Fanuc TP program (LS listing): FM171157.ls

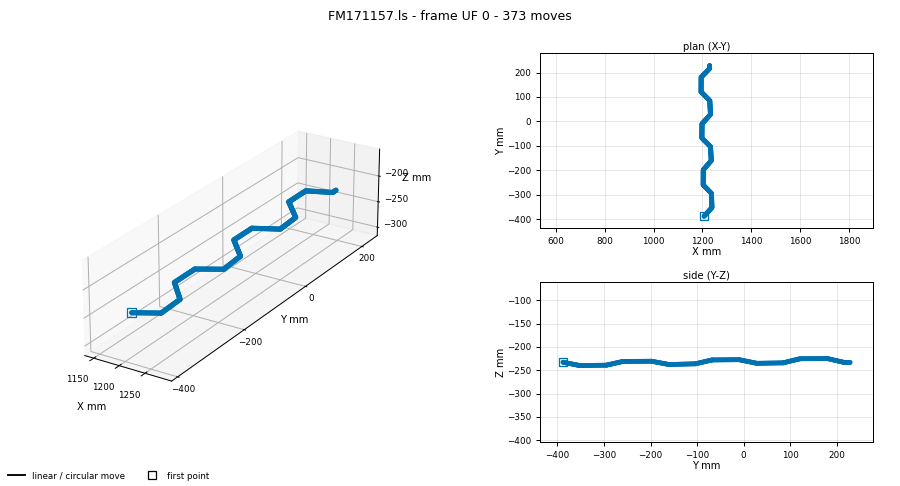
[picture p0: tool path of FM171157.ls in frame UF 0, 373 of 373 moves have a stored position in this frame; points joined in program order, loops and branches not executed]
/PROG  FM171157
/ATTR
OWNER		= MNEDITOR;
COMMENT		= "Auto FANUC move";
PROG_SIZE	= 0;
CREATE		= DATE 26-05-06  TIME 17:11:57;
MODIFIED	= DATE 26-05-06  TIME 17:11:57;
FILE_NAME	= ;
VERSION		= 0;
LINE_COUNT	= 378;
MEMORY_SIZE	= 0;
PROTECT		= READ_WRITE;
TCD:  STACK_SIZE	= 0,
      TASK_PRIORITY	= 50,
      TIME_SLICE	= 0,
      BUSY_LAMP_OFF	= 0,
      ABORT_REQUEST	= 0,
      PAUSE_REQUEST	= 0;
DEFAULT_GROUP	= 1,*,*,*,*;
CONTROL_CODE	= 00000000 00000000;
/MN
   1:  UFRAME_NUM=0 ;
   2:  UTOOL_NUM=1 ;
   3:  R[93]=10 ;
   4:  L P[1] 7mm/sec FINE ;
   5:  L P[2] 7mm/sec CNT50 ;
   6:  L P[3] 7mm/sec CNT50 ;
   7:  L P[4] 7mm/sec CNT50 ;
   8:  L P[5] 7mm/sec CNT50 ;
   9:  L P[6] 7mm/sec CNT50 ;
  10:  L P[7] 7mm/sec CNT50 ;
  11:  L P[8] 7mm/sec CNT50 ;
  12:  L P[9] 7mm/sec CNT50 ;
  13:  L P[10] 7mm/sec CNT50 ;
  14:  L P[11] 7mm/sec CNT50 ;
  15:  L P[12] 7mm/sec CNT50 ;
  16:  L P[13] 7mm/sec CNT50 ;
  17:  L P[14] 7mm/sec CNT50 ;
  18:  L P[15] 7mm/sec CNT50 ;
  19:  L P[16] 7mm/sec CNT50 ;
  20:  L P[17] 7mm/sec CNT50 ;
  21:  L P[18] 7mm/sec CNT50 ;
  22:  L P[19] 7mm/sec CNT50 ;
  23:  L P[20] 7mm/sec CNT50 ;
  24:  L P[21] 7mm/sec CNT50 ;
  25:  L P[22] 7mm/sec CNT50 ;
  26:  L P[23] 7mm/sec CNT50 ;
  27:  L P[24] 7mm/sec CNT50 ;
  28:  L P[25] 7mm/sec CNT50 ;
  29:  L P[26] 7mm/sec CNT50 ;
  30:  L P[27] 7mm/sec CNT50 ;
  31:  L P[28] 7mm/sec CNT50 ;
  32:  L P[29] 7mm/sec CNT50 ;
  33:  L P[30] 7mm/sec CNT50 ;
  34:  L P[31] 7mm/sec CNT50 ;
  35:  L P[32] 7mm/sec CNT50 ;
  36:  L P[33] 7mm/sec CNT50 ;
  37:  L P[34] 7mm/sec CNT50 ;
  38:  L P[35] 7mm/sec CNT50 ;
  39:  L P[36] 7mm/sec CNT50 ;
  40:  L P[37] 7mm/sec CNT50 ;
  41:  L P[38] 7mm/sec CNT50 ;
  42:  L P[39] 7mm/sec CNT50 ;
  43:  L P[40] 7mm/sec CNT50 ;
  44:  L P[41] 7mm/sec CNT50 ;
  45:  L P[42] 7mm/sec CNT50 ;
  46:  L P[43] 7mm/sec CNT50 ;
  47:  L P[44] 7mm/sec CNT50 ;
  48:  L P[45] 7mm/sec CNT50 ;
  49:  L P[46] 7mm/sec CNT50 ;
  50:  L P[47] 7mm/sec CNT50 ;
  51:  L P[48] 7mm/sec CNT50 ;
  52:  L P[49] 7mm/sec CNT50 ;
  53:  L P[50] 7mm/sec CNT50 ;
  54:  L P[51] 7mm/sec CNT50 ;
  55:  L P[52] 7mm/sec CNT50 ;
  56:  L P[53] 7mm/sec CNT50 ;
  57:  L P[54] 7mm/sec CNT50 ;
  58:  L P[55] 7mm/sec CNT50 ;
  59:  L P[56] 7mm/sec CNT50 ;
  60:  L P[57] 7mm/sec CNT50 ;
  61:  L P[58] 7mm/sec CNT50 ;
  62:  L P[59] 7mm/sec CNT50 ;
  63:  L P[60] 7mm/sec CNT50 ;
  64:  L P[61] 7mm/sec CNT50 ;
  65:  L P[62] 7mm/sec CNT50 ;
  66:  L P[63] 7mm/sec CNT50 ;
  67:  L P[64] 7mm/sec CNT50 ;
  68:  L P[65] 7mm/sec CNT50 ;
  69:  L P[66] 7mm/sec CNT50 ;
  70:  L P[67] 7mm/sec CNT50 ;
  71:  L P[68] 7mm/sec CNT50 ;
  72:  L P[69] 7mm/sec CNT50 ;
  73:  L P[70] 7mm/sec CNT50 ;
  74:  L P[71] 7mm/sec CNT50 ;
  75:  L P[72] 7mm/sec CNT50 ;
  76:  L P[73] 7mm/sec CNT50 ;
  77:  L P[74] 7mm/sec CNT50 ;
  78:  L P[75] 7mm/sec CNT50 ;
  79:  L P[76] 7mm/sec CNT50 ;
  80:  L P[77] 7mm/sec CNT50 ;
  81:  L P[78] 7mm/sec CNT50 ;
  82:  L P[79] 7mm/sec CNT50 ;
  83:  L P[80] 7mm/sec CNT50 ;
  84:  L P[81] 7mm/sec CNT50 ;
  85:  L P[82] 7mm/sec CNT50 ;
  86:  L P[83] 7mm/sec CNT50 ;
  87:  L P[84] 7mm/sec CNT50 ;
  88:  L P[85] 7mm/sec CNT50 ;
  89:  L P[86] 7mm/sec CNT50 ;
  90:  L P[87] 7mm/sec CNT50 ;
  91:  L P[88] 7mm/sec CNT50 ;
  92:  L P[89] 7mm/sec CNT50 ;
  93:  L P[90] 7mm/sec CNT50 ;
  94:  L P[91] 7mm/sec CNT50 ;
  95:  L P[92] 7mm/sec CNT50 ;
  96:  L P[93] 7mm/sec CNT50 ;
  97:  L P[94] 7mm/sec CNT50 ;
  98:  L P[95] 7mm/sec CNT50 ;
  99:  L P[96] 7mm/sec CNT50 ;
 100:  L P[97] 7mm/sec CNT50 ;
 101:  L P[98] 7mm/sec CNT50 ;
 102:  L P[99] 7mm/sec CNT50 ;
 103:  L P[100] 7mm/sec CNT50 ;
 104:  L P[101] 7mm/sec CNT50 ;
 105:  L P[102] 7mm/sec CNT50 ;
 106:  L P[103] 7mm/sec CNT50 ;
 107:  L P[104] 7mm/sec CNT50 ;
 108:  L P[105] 7mm/sec CNT50 ;
 109:  L P[106] 7mm/sec CNT50 ;
 110:  L P[107] 7mm/sec CNT50 ;
 111:  L P[108] 7mm/sec CNT50 ;
 112:  L P[109] 7mm/sec CNT50 ;
 113:  L P[110] 7mm/sec CNT50 ;
 114:  L P[111] 7mm/sec CNT50 ;
 115:  L P[112] 7mm/sec CNT50 ;
 116:  L P[113] 7mm/sec CNT50 ;
 117:  L P[114] 7mm/sec CNT50 ;
 118:  L P[115] 7mm/sec CNT50 ;
 119:  L P[116] 7mm/sec CNT50 ;
 120:  L P[117] 7mm/sec CNT50 ;
 121:  L P[118] 7mm/sec CNT50 ;
 122:  L P[119] 7mm/sec CNT50 ;
 123:  L P[120] 7mm/sec CNT50 ;
 124:  L P[121] 7mm/sec CNT50 ;
 125:  L P[122] 7mm/sec CNT50 ;
 126:  L P[123] 7mm/sec CNT50 ;
 127:  L P[124] 7mm/sec CNT50 ;
 128:  L P[125] 7mm/sec CNT50 ;
 129:  L P[126] 7mm/sec CNT50 ;
 130:  L P[127] 7mm/sec CNT50 ;
 131:  L P[128] 7mm/sec CNT50 ;
 132:  L P[129] 7mm/sec CNT50 ;
 133:  L P[130] 7mm/sec CNT50 ;
 134:  L P[131] 7mm/sec CNT50 ;
 135:  L P[132] 7mm/sec CNT50 ;
 136:  L P[133] 7mm/sec CNT50 ;
 137:  L P[134] 7mm/sec CNT50 ;
 138:  L P[135] 7mm/sec CNT50 ;
 139:  L P[136] 7mm/sec CNT50 ;
 140:  L P[137] 7mm/sec CNT50 ;
 141:  L P[138] 7mm/sec CNT50 ;
 142:  L P[139] 7mm/sec CNT50 ;
 143:  L P[140] 7mm/sec CNT50 ;
 144:  L P[141] 7mm/sec CNT50 ;
 145:  L P[142] 7mm/sec CNT50 ;
 146:  L P[143] 7mm/sec CNT50 ;
 147:  L P[144] 7mm/sec CNT50 ;
 148:  L P[145] 7mm/sec CNT50 ;
 149:  L P[146] 7mm/sec CNT50 ;
 150:  L P[147] 7mm/sec CNT50 ;
 151:  L P[148] 7mm/sec CNT50 ;
 152:  L P[149] 7mm/sec CNT50 ;
 153:  L P[150] 7mm/sec CNT50 ;
 154:  L P[151] 7mm/sec CNT50 ;
 155:  L P[152] 7mm/sec CNT50 ;
 156:  L P[153] 7mm/sec CNT50 ;
 157:  L P[154] 7mm/sec CNT50 ;
 158:  L P[155] 7mm/sec CNT50 ;
 159:  L P[156] 7mm/sec CNT50 ;
 160:  L P[157] 7mm/sec CNT50 ;
 161:  L P[158] 7mm/sec CNT50 ;
 162:  L P[159] 7mm/sec CNT50 ;
 163:  L P[160] 7mm/sec CNT50 ;
 164:  L P[161] 7mm/sec CNT50 ;
 165:  L P[162] 7mm/sec CNT50 ;
 166:  L P[163] 7mm/sec CNT50 ;
 167:  L P[164] 7mm/sec CNT50 ;
 168:  L P[165] 7mm/sec CNT50 ;
 169:  L P[166] 7mm/sec CNT50 ;
 170:  L P[167] 7mm/sec CNT50 ;
 171:  L P[168] 7mm/sec CNT50 ;
 172:  L P[169] 7mm/sec CNT50 ;
 173:  L P[170] 7mm/sec CNT50 ;
 174:  L P[171] 7mm/sec CNT50 ;
 175:  L P[172] 7mm/sec CNT50 ;
 176:  L P[173] 7mm/sec CNT50 ;
 177:  L P[174] 7mm/sec CNT50 ;
 178:  L P[175] 7mm/sec CNT50 ;
 179:  L P[176] 7mm/sec CNT50 ;
 180:  L P[177] 7mm/sec CNT50 ;
 181:  L P[178] 7mm/sec CNT50 ;
 182:  L P[179] 7mm/sec CNT50 ;
 183:  L P[180] 7mm/sec CNT50 ;
 184:  L P[181] 7mm/sec CNT50 ;
 185:  L P[182] 7mm/sec CNT50 ;
 186:  L P[183] 7mm/sec CNT50 ;
 187:  L P[184] 7mm/sec CNT50 ;
 188:  L P[185] 7mm/sec CNT50 ;
 189:  L P[186] 7mm/sec CNT50 ;
 190:  L P[187] 7mm/sec CNT50 ;
 191:  L P[188] 7mm/sec CNT50 ;
 192:  L P[189] 7mm/sec CNT50 ;
 193:  L P[190] 7mm/sec CNT50 ;
 194:  L P[191] 7mm/sec CNT50 ;
 195:  L P[192] 7mm/sec CNT50 ;
 196:  L P[193] 7mm/sec CNT50 ;
 197:  L P[194] 7mm/sec CNT50 ;
 198:  L P[195] 7mm/sec CNT50 ;
 199:  L P[196] 7mm/sec CNT50 ;
 200:  L P[197] 7mm/sec CNT50 ;
 201:  L P[198] 7mm/sec CNT50 ;
 202:  L P[199] 7mm/sec CNT50 ;
 203:  L P[200] 7mm/sec CNT50 ;
 204:  L P[201] 7mm/sec CNT50 ;
 205:  L P[202] 7mm/sec CNT50 ;
 206:  L P[203] 7mm/sec CNT50 ;
 207:  L P[204] 7mm/sec CNT50 ;
 208:  L P[205] 7mm/sec CNT50 ;
 209:  L P[206] 7mm/sec CNT50 ;
 210:  L P[207] 7mm/sec CNT50 ;
 211:  L P[208] 7mm/sec CNT50 ;
 212:  L P[209] 7mm/sec CNT50 ;
 213:  L P[210] 7mm/sec CNT50 ;
 214:  L P[211] 7mm/sec CNT50 ;
 215:  L P[212] 7mm/sec CNT50 ;
 216:  L P[213] 7mm/sec CNT50 ;
 217:  L P[214] 7mm/sec CNT50 ;
 218:  L P[215] 7mm/sec CNT50 ;
 219:  L P[216] 7mm/sec CNT50 ;
 220:  L P[217] 7mm/sec CNT50 ;
 221:  L P[218] 7mm/sec CNT50 ;
 222:  L P[219] 7mm/sec CNT50 ;
 223:  L P[220] 7mm/sec CNT50 ;
 224:  L P[221] 7mm/sec CNT50 ;
 225:  L P[222] 7mm/sec CNT50 ;
 226:  L P[223] 7mm/sec CNT50 ;
 227:  L P[224] 7mm/sec CNT50 ;
 228:  L P[225] 7mm/sec CNT50 ;
 229:  L P[226] 7mm/sec CNT50 ;
 230:  L P[227] 7mm/sec CNT50 ;
 231:  L P[228] 7mm/sec CNT50 ;
 232:  L P[229] 7mm/sec CNT50 ;
 233:  L P[230] 7mm/sec CNT50 ;
 234:  L P[231] 7mm/sec CNT50 ;
 235:  L P[232] 7mm/sec CNT50 ;
 236:  L P[233] 7mm/sec CNT50 ;
 237:  L P[234] 7mm/sec CNT50 ;
 238:  L P[235] 7mm/sec CNT50 ;
 239:  L P[236] 7mm/sec CNT50 ;
 240:  L P[237] 7mm/sec CNT50 ;
 241:  L P[238] 7mm/sec CNT50 ;
 242:  L P[239] 7mm/sec CNT50 ;
 243:  L P[240] 7mm/sec CNT50 ;
 244:  L P[241] 7mm/sec CNT50 ;
 245:  L P[242] 7mm/sec CNT50 ;
 246:  L P[243] 7mm/sec CNT50 ;
 247:  L P[244] 7mm/sec CNT50 ;
 248:  L P[245] 7mm/sec CNT50 ;
 249:  L P[246] 7mm/sec CNT50 ;
 250:  L P[247] 7mm/sec CNT50 ;
 251:  L P[248] 7mm/sec CNT50 ;
 252:  L P[249] 7mm/sec CNT50 ;
 253:  L P[250] 7mm/sec CNT50 ;
 254:  L P[251] 7mm/sec CNT50 ;
 255:  L P[252] 7mm/sec CNT50 ;
 256:  L P[253] 7mm/sec CNT50 ;
 257:  L P[254] 7mm/sec CNT50 ;
 258:  L P[255] 7mm/sec CNT50 ;
 259:  L P[256] 7mm/sec CNT50 ;
 260:  L P[257] 7mm/sec CNT50 ;
 261:  L P[258] 7mm/sec CNT50 ;
 262:  L P[259] 7mm/sec CNT50 ;
 263:  L P[260] 7mm/sec CNT50 ;
 264:  L P[261] 7mm/sec CNT50 ;
 265:  L P[262] 7mm/sec CNT50 ;
 266:  L P[263] 7mm/sec CNT50 ;
 267:  L P[264] 7mm/sec CNT50 ;
 268:  L P[265] 7mm/sec CNT50 ;
 269:  L P[266] 7mm/sec CNT50 ;
 270:  L P[267] 7mm/sec CNT50 ;
 271:  L P[268] 7mm/sec CNT50 ;
 272:  L P[269] 7mm/sec CNT50 ;
 273:  L P[270] 7mm/sec CNT50 ;
 274:  L P[271] 7mm/sec CNT50 ;
 275:  L P[272] 7mm/sec CNT50 ;
 276:  L P[273] 7mm/sec CNT50 ;
 277:  L P[274] 7mm/sec CNT50 ;
 278:  L P[275] 7mm/sec CNT50 ;
 279:  L P[276] 7mm/sec CNT50 ;
 280:  L P[277] 7mm/sec CNT50 ;
 281:  L P[278] 7mm/sec CNT50 ;
 282:  L P[279] 7mm/sec CNT50 ;
 283:  L P[280] 7mm/sec CNT50 ;
 284:  L P[281] 7mm/sec CNT50 ;
 285:  L P[282] 7mm/sec CNT50 ;
 286:  L P[283] 7mm/sec CNT50 ;
 287:  L P[284] 7mm/sec CNT50 ;
 288:  L P[285] 7mm/sec CNT50 ;
 289:  L P[286] 7mm/sec CNT50 ;
 290:  L P[287] 7mm/sec CNT50 ;
 291:  L P[288] 7mm/sec CNT50 ;
 292:  L P[289] 7mm/sec CNT50 ;
 293:  L P[290] 7mm/sec CNT50 ;
 294:  L P[291] 7mm/sec CNT50 ;
 295:  L P[292] 7mm/sec CNT50 ;
 296:  L P[293] 7mm/sec CNT50 ;
 297:  L P[294] 7mm/sec CNT50 ;
 298:  L P[295] 7mm/sec CNT50 ;
 299:  L P[296] 7mm/sec CNT50 ;
 300:  L P[297] 7mm/sec CNT50 ;
 301:  L P[298] 7mm/sec CNT50 ;
 302:  L P[299] 7mm/sec CNT50 ;
 303:  L P[300] 7mm/sec CNT50 ;
 304:  L P[301] 7mm/sec CNT50 ;
 305:  L P[302] 7mm/sec CNT50 ;
 306:  L P[303] 7mm/sec CNT50 ;
 307:  L P[304] 7mm/sec CNT50 ;
 308:  L P[305] 7mm/sec CNT50 ;
 309:  L P[306] 7mm/sec CNT50 ;
 310:  L P[307] 7mm/sec CNT50 ;
 311:  L P[308] 7mm/sec CNT50 ;
 312:  L P[309] 7mm/sec CNT50 ;
 313:  L P[310] 7mm/sec CNT50 ;
 314:  L P[311] 7mm/sec CNT50 ;
 315:  L P[312] 7mm/sec CNT50 ;
 316:  L P[313] 7mm/sec CNT50 ;
 317:  L P[314] 7mm/sec CNT50 ;
 318:  L P[315] 7mm/sec CNT50 ;
 319:  L P[316] 7mm/sec CNT50 ;
 320:  L P[317] 7mm/sec CNT50 ;
 321:  L P[318] 7mm/sec CNT50 ;
 322:  L P[319] 7mm/sec CNT50 ;
 323:  L P[320] 7mm/sec CNT50 ;
 324:  L P[321] 7mm/sec CNT50 ;
 325:  L P[322] 7mm/sec CNT50 ;
 326:  L P[323] 7mm/sec CNT50 ;
 327:  L P[324] 7mm/sec CNT50 ;
 328:  L P[325] 7mm/sec CNT50 ;
 329:  L P[326] 7mm/sec CNT50 ;
 330:  L P[327] 7mm/sec CNT50 ;
 331:  L P[328] 7mm/sec CNT50 ;
 332:  L P[329] 7mm/sec CNT50 ;
 333:  L P[330] 7mm/sec CNT50 ;
 334:  L P[331] 7mm/sec CNT50 ;
 335:  L P[332] 7mm/sec CNT50 ;
 336:  L P[333] 7mm/sec CNT50 ;
 337:  L P[334] 7mm/sec CNT50 ;
 338:  L P[335] 7mm/sec CNT50 ;
 339:  L P[336] 7mm/sec CNT50 ;
 340:  L P[337] 7mm/sec CNT50 ;
 341:  L P[338] 7mm/sec CNT50 ;
 342:  L P[339] 7mm/sec CNT50 ;
 343:  L P[340] 7mm/sec CNT50 ;
 344:  L P[341] 7mm/sec CNT50 ;
 345:  L P[342] 7mm/sec CNT50 ;
 346:  L P[343] 7mm/sec CNT50 ;
 347:  L P[344] 7mm/sec CNT50 ;
 348:  L P[345] 7mm/sec CNT50 ;
 349:  L P[346] 7mm/sec CNT50 ;
 350:  L P[347] 7mm/sec CNT50 ;
 351:  L P[348] 7mm/sec CNT50 ;
 352:  L P[349] 7mm/sec CNT50 ;
 353:  L P[350] 7mm/sec CNT50 ;
 354:  L P[351] 7mm/sec CNT50 ;
 355:  L P[352] 7mm/sec CNT50 ;
 356:  L P[353] 7mm/sec CNT50 ;
 357:  L P[354] 7mm/sec CNT50 ;
 358:  L P[355] 7mm/sec CNT50 ;
 359:  L P[356] 7mm/sec CNT50 ;
 360:  L P[357] 7mm/sec CNT50 ;
 361:  L P[358] 7mm/sec CNT50 ;
 362:  L P[359] 7mm/sec CNT50 ;
 363:  L P[360] 7mm/sec CNT50 ;
 364:  L P[361] 7mm/sec CNT50 ;
 365:  L P[362] 7mm/sec CNT50 ;
 366:  L P[363] 7mm/sec CNT50 ;
 367:  L P[364] 7mm/sec CNT50 ;
 368:  L P[365] 7mm/sec CNT50 ;
 369:  L P[366] 7mm/sec CNT50 ;
 370:  L P[367] 7mm/sec CNT50 ;
 371:  L P[368] 7mm/sec CNT50 ;
 372:  L P[369] 7mm/sec CNT50 ;
 373:  L P[370] 7mm/sec CNT50 ;
 374:  L P[371] 7mm/sec CNT50 ;
 375:  L P[372] 7mm/sec CNT50 ;
 376:  L P[373] 7mm/sec FINE ;
 377:  R[93]=1 ;
 378:  END ;
/POS
P[1]{
   GP1:
	UF : 0, UT : 1,		CONFIG : 'N U T, 0, 0, 0',
	X = 1206.347  mm,	Y = -388.199  mm,	Z = -232.788  mm,
	W = 0.000 deg,	P = 30.000 deg,	R = 160.000 deg
};
P[2]{
   GP1:
	UF : 0, UT : 1,		CONFIG : 'N U T, 0, 0, 0',
	X = 1207.673  mm,	Y = -386.730  mm,	Z = -233.078  mm,
	W = 0.000 deg,	P = 30.000 deg,	R = 160.000 deg
};
P[3]{
   GP1:
	UF : 0, UT : 1,		CONFIG : 'N U T, 0, 0, 0',
	X = 1208.999  mm,	Y = -385.261  mm,	Z = -233.367  mm,
	W = 0.000 deg,	P = 30.000 deg,	R = 160.000 deg
};
P[4]{
   GP1:
	UF : 0, UT : 1,		CONFIG : 'N U T, 0, 0, 0',
	X = 1210.325  mm,	Y = -383.791  mm,	Z = -233.656  mm,
	W = 0.000 deg,	P = 30.000 deg,	R = 160.000 deg
};
P[5]{
   GP1:
	UF : 0, UT : 1,		CONFIG : 'N U T, 0, 0, 0',
	X = 1211.651  mm,	Y = -382.322  mm,	Z = -233.946  mm,
	W = 0.000 deg,	P = 30.000 deg,	R = 160.000 deg
};
P[6]{
   GP1:
	UF : 0, UT : 1,		CONFIG : 'N U T, 0, 0, 0',
	X = 1212.977  mm,	Y = -380.853  mm,	Z = -234.235  mm,
	W = 0.000 deg,	P = 30.000 deg,	R = 160.000 deg
};
P[7]{
   GP1:
	UF : 0, UT : 1,		CONFIG : 'N U T, 0, 0, 0',
	X = 1214.303  mm,	Y = -379.384  mm,	Z = -234.524  mm,
	W = 0.000 deg,	P = 30.000 deg,	R = 160.000 deg
};
P[8]{
   GP1:
	UF : 0, UT : 1,		CONFIG : 'N U T, 0, 0, 0',
	X = 1215.629  mm,	Y = -377.915  mm,	Z = -234.814  mm,
	W = 0.000 deg,	P = 30.000 deg,	R = 160.000 deg
};
P[9]{
   GP1:
	UF : 0, UT : 1,		CONFIG : 'N U T, 0, 0, 0',
	X = 1216.955  mm,	Y = -376.446  mm,	Z = -235.103  mm,
	W = 0.000 deg,	P = 30.000 deg,	R = 160.000 deg
};
P[10]{
   GP1:
	UF : 0, UT : 1,		CONFIG : 'N U T, 0, 0, 0',
	X = 1218.281  mm,	Y = -374.977  mm,	Z = -235.392  mm,
	W = 0.000 deg,	P = 30.000 deg,	R = 160.000 deg
};
P[11]{
   GP1:
	UF : 0, UT : 1,		CONFIG : 'N U T, 0, 0, 0',
	X = 1219.607  mm,	Y = -373.508  mm,	Z = -235.682  mm,
	W = 0.000 deg,	P = 30.000 deg,	R = 160.000 deg
};
P[12]{
   GP1:
	UF : 0, UT : 1,		CONFIG : 'N U T, 0, 0, 0',
	X = 1220.933  mm,	Y = -372.039  mm,	Z = -235.971  mm,
	W = 0.000 deg,	P = 30.000 deg,	R = 160.000 deg
};
P[13]{
   GP1:
	UF : 0, UT : 1,		CONFIG : 'N U T, 0, 0, 0',
	X = 1222.258  mm,	Y = -370.570  mm,	Z = -236.260  mm,
	W = 0.000 deg,	P = 30.000 deg,	R = 160.000 deg
};
P[14]{
   GP1:
	UF : 0, UT : 1,		CONFIG : 'N U T, 0, 0, 0',
	X = 1223.584  mm,	Y = -369.101  mm,	Z = -236.549  mm,
	W = 0.000 deg,	P = 30.000 deg,	R = 160.000 deg
};
P[15]{
   GP1:
	UF : 0, UT : 1,		CONFIG : 'N U T, 0, 0, 0',
	X = 1224.910  mm,	Y = -367.632  mm,	Z = -236.839  mm,
	W = 0.000 deg,	P = 30.000 deg,	R = 160.000 deg
};
P[16]{
   GP1:
	UF : 0, UT : 1,		CONFIG : 'N U T, 0, 0, 0',
	X = 1226.236  mm,	Y = -366.163  mm,	Z = -237.128  mm,
	W = 0.000 deg,	P = 30.000 deg,	R = 160.000 deg
};
P[17]{
   GP1:
	UF : 0, UT : 1,		CONFIG : 'N U T, 0, 0, 0',
	X = 1227.562  mm,	Y = -364.694  mm,	Z = -237.417  mm,
	W = 0.000 deg,	P = 30.000 deg,	R = 160.000 deg
};
P[18]{
   GP1:
	UF : 0, UT : 1,		CONFIG : 'N U T, 0, 0, 0',
	X = 1228.888  mm,	Y = -363.225  mm,	Z = -237.707  mm,
	W = 0.000 deg,	P = 30.000 deg,	R = 160.000 deg
};
P[19]{
   GP1:
	UF : 0, UT : 1,		CONFIG : 'N U T, 0, 0, 0',
	X = 1230.214  mm,	Y = -361.756  mm,	Z = -237.996  mm,
	W = 0.000 deg,	P = 30.000 deg,	R = 160.000 deg
};
P[20]{
   GP1:
	UF : 0, UT : 1,		CONFIG : 'N U T, 0, 0, 0',
	X = 1231.540  mm,	Y = -360.287  mm,	Z = -238.285  mm,
	W = 0.000 deg,	P = 30.000 deg,	R = 160.000 deg
};
P[21]{
   GP1:
	UF : 0, UT : 1,		CONFIG : 'N U T, 0, 0, 0',
	X = 1232.866  mm,	Y = -358.818  mm,	Z = -238.575  mm,
	W = 0.000 deg,	P = 30.000 deg,	R = 164.342 deg
};
P[22]{
   GP1:
	UF : 0, UT : 1,		CONFIG : 'N U T, 0, 0, 0',
	X = 1234.192  mm,	Y = -357.349  mm,	Z = -238.864  mm,
	W = 0.000 deg,	P = 30.000 deg,	R = 168.685 deg
};
P[23]{
   GP1:
	UF : 0, UT : 1,		CONFIG : 'N U T, 0, 0, 0',
	X = 1235.518  mm,	Y = -355.880  mm,	Z = -239.153  mm,
	W = 0.000 deg,	P = 30.000 deg,	R = 173.027 deg
};
P[24]{
   GP1:
	UF : 0, UT : 1,		CONFIG : 'N U T, 0, 0, 0',
	X = 1236.844  mm,	Y = -354.410  mm,	Z = -239.443  mm,
	W = 0.000 deg,	P = 30.000 deg,	R = 177.369 deg
};
P[25]{
   GP1:
	UF : 0, UT : 1,		CONFIG : 'N U T, 0, 0, 0',
	X = 1238.170  mm,	Y = -352.941  mm,	Z = -239.732  mm,
	W = 0.000 deg,	P = 30.000 deg,	R = -178.289 deg
};
P[26]{
   GP1:
	UF : 0, UT : 1,		CONFIG : 'N U T, 0, 0, 0',
	X = 1238.798  mm,	Y = -352.246  mm,	Z = -239.869  mm,
	W = 0.000 deg,	P = 30.000 deg,	R = -178.289 deg
};
P[27]{
   GP1:
	UF : 0, UT : 1,		CONFIG : 'N U T, 0, 0, 0',
	X = 1238.766  mm,	Y = -351.193  mm,	Z = -239.854  mm,
	W = 0.000 deg,	P = 30.000 deg,	R = -178.289 deg
};
P[28]{
   GP1:
	UF : 0, UT : 1,		CONFIG : 'N U T, 0, 0, 0',
	X = 1238.706  mm,	Y = -349.194  mm,	Z = -239.826  mm,
	W = 0.000 deg,	P = 30.000 deg,	R = -178.289 deg
};
P[29]{
   GP1:
	UF : 0, UT : 1,		CONFIG : 'N U T, 0, 0, 0',
	X = 1238.647  mm,	Y = -347.195  mm,	Z = -239.798  mm,
	W = 0.000 deg,	P = 30.000 deg,	R = -178.289 deg
};
P[30]{
   GP1:
	UF : 0, UT : 1,		CONFIG : 'N U T, 0, 0, 0',
	X = 1238.587  mm,	Y = -345.197  mm,	Z = -239.769  mm,
	W = 0.000 deg,	P = 30.000 deg,	R = -178.289 deg
};
P[31]{
   GP1:
	UF : 0, UT : 1,		CONFIG : 'N U T, 0, 0, 0',
	X = 1238.527  mm,	Y = -343.198  mm,	Z = -239.741  mm,
	W = 0.000 deg,	P = 30.000 deg,	R = -178.289 deg
};
P[32]{
   GP1:
	UF : 0, UT : 1,		CONFIG : 'N U T, 0, 0, 0',
	X = 1238.468  mm,	Y = -341.199  mm,	Z = -239.713  mm,
	W = 0.000 deg,	P = 30.000 deg,	R = -178.289 deg
};
P[33]{
   GP1:
	UF : 0, UT : 1,		CONFIG : 'N U T, 0, 0, 0',
	X = 1238.408  mm,	Y = -339.200  mm,	Z = -239.685  mm,
	W = 0.000 deg,	P = 30.000 deg,	R = -178.289 deg
};
P[34]{
   GP1:
	UF : 0, UT : 1,		CONFIG : 'N U T, 0, 0, 0',
	X = 1238.348  mm,	Y = -337.201  mm,	Z = -239.656  mm,
	W = 0.000 deg,	P = 30.000 deg,	R = -178.289 deg
};
P[35]{
   GP1:
	UF : 0, UT : 1,		CONFIG : 'N U T, 0, 0, 0',
	X = 1238.288  mm,	Y = -335.202  mm,	Z = -239.628  mm,
	W = 0.000 deg,	P = 30.000 deg,	R = -178.289 deg
};
P[36]{
   GP1:
	UF : 0, UT : 1,		CONFIG : 'N U T, 0, 0, 0',
	X = 1238.229  mm,	Y = -333.203  mm,	Z = -239.600  mm,
	W = 0.000 deg,	P = 30.000 deg,	R = -178.289 deg
};
P[37]{
   GP1:
	UF : 0, UT : 1,		CONFIG : 'N U T, 0, 0, 0',
	X = 1238.169  mm,	Y = -331.204  mm,	Z = -239.572  mm,
	W = 0.000 deg,	P = 30.000 deg,	R = -178.289 deg
};
P[38]{
   GP1:
	UF : 0, UT : 1,		CONFIG : 'N U T, 0, 0, 0',
	X = 1238.109  mm,	Y = -329.205  mm,	Z = -239.543  mm,
	W = 0.000 deg,	P = 30.000 deg,	R = -178.289 deg
};
P[39]{
   GP1:
	UF : 0, UT : 1,		CONFIG : 'N U T, 0, 0, 0',
	X = 1238.049  mm,	Y = -327.206  mm,	Z = -239.515  mm,
	W = 0.000 deg,	P = 30.000 deg,	R = -178.289 deg
};
P[40]{
   GP1:
	UF : 0, UT : 1,		CONFIG : 'N U T, 0, 0, 0',
	X = 1237.990  mm,	Y = -325.207  mm,	Z = -239.487  mm,
	W = 0.000 deg,	P = 30.000 deg,	R = -178.289 deg
};
P[41]{
   GP1:
	UF : 0, UT : 1,		CONFIG : 'N U T, 0, 0, 0',
	X = 1237.930  mm,	Y = -323.209  mm,	Z = -239.459  mm,
	W = 0.000 deg,	P = 30.000 deg,	R = -178.289 deg
};
P[42]{
   GP1:
	UF : 0, UT : 1,		CONFIG : 'N U T, 0, 0, 0',
	X = 1237.870  mm,	Y = -321.210  mm,	Z = -239.431  mm,
	W = 0.000 deg,	P = 30.000 deg,	R = -178.289 deg
};
P[43]{
   GP1:
	UF : 0, UT : 1,		CONFIG : 'N U T, 0, 0, 0',
	X = 1237.811  mm,	Y = -319.211  mm,	Z = -239.402  mm,
	W = 0.000 deg,	P = 30.000 deg,	R = -178.289 deg
};
P[44]{
   GP1:
	UF : 0, UT : 1,		CONFIG : 'N U T, 0, 0, 0',
	X = 1237.751  mm,	Y = -317.212  mm,	Z = -239.374  mm,
	W = 0.000 deg,	P = 30.000 deg,	R = -178.289 deg
};
P[45]{
   GP1:
	UF : 0, UT : 1,		CONFIG : 'N U T, 0, 0, 0',
	X = 1237.691  mm,	Y = -315.213  mm,	Z = -239.346  mm,
	W = 0.000 deg,	P = 30.000 deg,	R = -178.289 deg
};
P[46]{
   GP1:
	UF : 0, UT : 1,		CONFIG : 'N U T, 0, 0, 0',
	X = 1237.631  mm,	Y = -313.214  mm,	Z = -239.318  mm,
	W = 0.000 deg,	P = 30.000 deg,	R = -178.289 deg
};
P[47]{
   GP1:
	UF : 0, UT : 1,		CONFIG : 'N U T, 0, 0, 0',
	X = 1237.572  mm,	Y = -311.215  mm,	Z = -239.289  mm,
	W = 0.000 deg,	P = 30.000 deg,	R = -178.289 deg
};
P[48]{
   GP1:
	UF : 0, UT : 1,		CONFIG : 'N U T, 0, 0, 0',
	X = 1237.512  mm,	Y = -309.216  mm,	Z = -239.261  mm,
	W = 0.000 deg,	P = 30.000 deg,	R = -178.289 deg
};
P[49]{
   GP1:
	UF : 0, UT : 1,		CONFIG : 'N U T, 0, 0, 0',
	X = 1237.452  mm,	Y = -307.217  mm,	Z = -239.233  mm,
	W = 0.000 deg,	P = 30.000 deg,	R = -178.289 deg
};
P[50]{
   GP1:
	UF : 0, UT : 1,		CONFIG : 'N U T, 0, 0, 0',
	X = 1237.393  mm,	Y = -305.218  mm,	Z = -239.205  mm,
	W = 0.000 deg,	P = 30.000 deg,	R = -178.289 deg
};
P[51]{
   GP1:
	UF : 0, UT : 1,		CONFIG : 'N U T, 0, 0, 0',
	X = 1237.333  mm,	Y = -303.219  mm,	Z = -239.177  mm,
	W = 0.000 deg,	P = 30.000 deg,	R = -172.704 deg
};
P[52]{
   GP1:
	UF : 0, UT : 1,		CONFIG : 'N U T, 0, 0, 0',
	X = 1237.273  mm,	Y = -301.221  mm,	Z = -239.148  mm,
	W = 0.000 deg,	P = 30.000 deg,	R = -169.047 deg
};
P[53]{
   GP1:
	UF : 0, UT : 1,		CONFIG : 'N U T, 0, 0, 0',
	X = 1237.213  mm,	Y = -299.222  mm,	Z = -239.120  mm,
	W = 0.000 deg,	P = 30.000 deg,	R = -165.389 deg
};
P[54]{
   GP1:
	UF : 0, UT : 1,		CONFIG : 'N U T, 0, 0, 0',
	X = 1237.154  mm,	Y = -297.223  mm,	Z = -239.092  mm,
	W = 0.000 deg,	P = 30.000 deg,	R = -161.731 deg
};
P[55]{
   GP1:
	UF : 0, UT : 1,		CONFIG : 'N U T, 0, 0, 0',
	X = 1237.094  mm,	Y = -295.224  mm,	Z = -239.064  mm,
	W = 0.000 deg,	P = 30.000 deg,	R = -160.000 deg
};
P[56]{
   GP1:
	UF : 0, UT : 1,		CONFIG : 'N U T, 0, 0, 0',
	X = 1237.079  mm,	Y = -294.716  mm,	Z = -239.056  mm,
	W = 0.000 deg,	P = 30.000 deg,	R = -160.000 deg
};
P[57]{
   GP1:
	UF : 0, UT : 1,		CONFIG : 'N U T, 0, 0, 0',
	X = 1236.053  mm,	Y = -293.659  mm,	Z = -238.818  mm,
	W = 0.000 deg,	P = 30.000 deg,	R = -160.000 deg
};
P[58]{
   GP1:
	UF : 0, UT : 1,		CONFIG : 'N U T, 0, 0, 0',
	X = 1234.678  mm,	Y = -292.243  mm,	Z = -238.498  mm,
	W = 0.000 deg,	P = 30.000 deg,	R = -160.000 deg
};
P[59]{
   GP1:
	UF : 0, UT : 1,		CONFIG : 'N U T, 0, 0, 0',
	X = 1233.303  mm,	Y = -290.826  mm,	Z = -238.177  mm,
	W = 0.000 deg,	P = 30.000 deg,	R = -160.000 deg
};
P[60]{
   GP1:
	UF : 0, UT : 1,		CONFIG : 'N U T, 0, 0, 0',
	X = 1231.928  mm,	Y = -289.409  mm,	Z = -237.857  mm,
	W = 0.000 deg,	P = 30.000 deg,	R = -160.000 deg
};
P[61]{
   GP1:
	UF : 0, UT : 1,		CONFIG : 'N U T, 0, 0, 0',
	X = 1230.553  mm,	Y = -287.992  mm,	Z = -237.537  mm,
	W = 0.000 deg,	P = 30.000 deg,	R = -160.000 deg
};
P[62]{
   GP1:
	UF : 0, UT : 1,		CONFIG : 'N U T, 0, 0, 0',
	X = 1229.179  mm,	Y = -286.575  mm,	Z = -237.217  mm,
	W = 0.000 deg,	P = 30.000 deg,	R = -160.000 deg
};
P[63]{
   GP1:
	UF : 0, UT : 1,		CONFIG : 'N U T, 0, 0, 0',
	X = 1227.804  mm,	Y = -285.159  mm,	Z = -236.897  mm,
	W = 0.000 deg,	P = 30.000 deg,	R = -160.000 deg
};
P[64]{
   GP1:
	UF : 0, UT : 1,		CONFIG : 'N U T, 0, 0, 0',
	X = 1226.429  mm,	Y = -283.742  mm,	Z = -236.577  mm,
	W = 0.000 deg,	P = 30.000 deg,	R = -160.000 deg
};
P[65]{
   GP1:
	UF : 0, UT : 1,		CONFIG : 'N U T, 0, 0, 0',
	X = 1225.054  mm,	Y = -282.325  mm,	Z = -236.257  mm,
	W = 0.000 deg,	P = 30.000 deg,	R = -160.000 deg
};
P[66]{
   GP1:
	UF : 0, UT : 1,		CONFIG : 'N U T, 0, 0, 0',
	X = 1223.679  mm,	Y = -280.908  mm,	Z = -235.937  mm,
	W = 0.000 deg,	P = 30.000 deg,	R = -160.000 deg
};
P[67]{
   GP1:
	UF : 0, UT : 1,		CONFIG : 'N U T, 0, 0, 0',
	X = 1222.304  mm,	Y = -279.491  mm,	Z = -235.617  mm,
	W = 0.000 deg,	P = 30.000 deg,	R = -160.000 deg
};
P[68]{
   GP1:
	UF : 0, UT : 1,		CONFIG : 'N U T, 0, 0, 0',
	X = 1220.929  mm,	Y = -278.075  mm,	Z = -235.297  mm,
	W = 0.000 deg,	P = 30.000 deg,	R = -160.000 deg
};
P[69]{
   GP1:
	UF : 0, UT : 1,		CONFIG : 'N U T, 0, 0, 0',
	X = 1219.554  mm,	Y = -276.658  mm,	Z = -234.977  mm,
	W = 0.000 deg,	P = 30.000 deg,	R = -160.000 deg
};
P[70]{
   GP1:
	UF : 0, UT : 1,		CONFIG : 'N U T, 0, 0, 0',
	X = 1218.180  mm,	Y = -275.241  mm,	Z = -234.656  mm,
	W = 0.000 deg,	P = 30.000 deg,	R = -160.000 deg
};
P[71]{
   GP1:
	UF : 0, UT : 1,		CONFIG : 'N U T, 0, 0, 0',
	X = 1216.805  mm,	Y = -273.824  mm,	Z = -234.336  mm,
	W = 0.000 deg,	P = 30.000 deg,	R = -160.000 deg
};
P[72]{
   GP1:
	UF : 0, UT : 1,		CONFIG : 'N U T, 0, 0, 0',
	X = 1215.430  mm,	Y = -272.408  mm,	Z = -234.016  mm,
	W = 0.000 deg,	P = 30.000 deg,	R = -160.000 deg
};
P[73]{
   GP1:
	UF : 0, UT : 1,		CONFIG : 'N U T, 0, 0, 0',
	X = 1214.055  mm,	Y = -270.991  mm,	Z = -233.696  mm,
	W = 0.000 deg,	P = 30.000 deg,	R = -160.000 deg
};
P[74]{
   GP1:
	UF : 0, UT : 1,		CONFIG : 'N U T, 0, 0, 0',
	X = 1212.680  mm,	Y = -269.574  mm,	Z = -233.376  mm,
	W = 0.000 deg,	P = 30.000 deg,	R = -160.000 deg
};
P[75]{
   GP1:
	UF : 0, UT : 1,		CONFIG : 'N U T, 0, 0, 0',
	X = 1211.305  mm,	Y = -268.157  mm,	Z = -233.056  mm,
	W = 0.000 deg,	P = 30.000 deg,	R = -160.000 deg
};
P[76]{
   GP1:
	UF : 0, UT : 1,		CONFIG : 'N U T, 0, 0, 0',
	X = 1209.930  mm,	Y = -266.740  mm,	Z = -232.736  mm,
	W = 0.000 deg,	P = 30.000 deg,	R = -160.000 deg
};
P[77]{
   GP1:
	UF : 0, UT : 1,		CONFIG : 'N U T, 0, 0, 0',
	X = 1208.555  mm,	Y = -265.324  mm,	Z = -232.416  mm,
	W = 0.000 deg,	P = 30.000 deg,	R = -167.071 deg
};
P[78]{
   GP1:
	UF : 0, UT : 1,		CONFIG : 'N U T, 0, 0, 0',
	X = 1207.181  mm,	Y = -263.907  mm,	Z = -232.096  mm,
	W = 0.000 deg,	P = 30.000 deg,	R = -171.121 deg
};
P[79]{
   GP1:
	UF : 0, UT : 1,		CONFIG : 'N U T, 0, 0, 0',
	X = 1205.806  mm,	Y = -262.490  mm,	Z = -231.776  mm,
	W = 0.000 deg,	P = 30.000 deg,	R = -175.171 deg
};
P[80]{
   GP1:
	UF : 0, UT : 1,		CONFIG : 'N U T, 0, 0, 0',
	X = 1204.431  mm,	Y = -261.073  mm,	Z = -231.455  mm,
	W = 0.000 deg,	P = 30.000 deg,	R = -179.220 deg
};
P[81]{
   GP1:
	UF : 0, UT : 1,		CONFIG : 'N U T, 0, 0, 0',
	X = 1203.056  mm,	Y = -259.657  mm,	Z = -231.135  mm,
	W = 0.000 deg,	P = 30.000 deg,	R = 179.752 deg
};
P[82]{
   GP1:
	UF : 0, UT : 1,		CONFIG : 'N U T, 0, 0, 0',
	X = 1202.896  mm,	Y = -259.492  mm,	Z = -231.098  mm,
	W = 0.000 deg,	P = 30.000 deg,	R = 179.752 deg
};
P[83]{
   GP1:
	UF : 0, UT : 1,		CONFIG : 'N U T, 0, 0, 0',
	X = 1202.904  mm,	Y = -257.724  mm,	Z = -231.083  mm,
	W = 0.000 deg,	P = 30.000 deg,	R = 179.752 deg
};
P[84]{
   GP1:
	UF : 0, UT : 1,		CONFIG : 'N U T, 0, 0, 0',
	X = 1202.912  mm,	Y = -255.725  mm,	Z = -231.067  mm,
	W = 0.000 deg,	P = 30.000 deg,	R = 179.752 deg
};
P[85]{
   GP1:
	UF : 0, UT : 1,		CONFIG : 'N U T, 0, 0, 0',
	X = 1202.921  mm,	Y = -253.725  mm,	Z = -231.050  mm,
	W = 0.000 deg,	P = 30.000 deg,	R = 179.752 deg
};
P[86]{
   GP1:
	UF : 0, UT : 1,		CONFIG : 'N U T, 0, 0, 0',
	X = 1202.930  mm,	Y = -251.725  mm,	Z = -231.033  mm,
	W = 0.000 deg,	P = 30.000 deg,	R = 179.752 deg
};
P[87]{
   GP1:
	UF : 0, UT : 1,		CONFIG : 'N U T, 0, 0, 0',
	X = 1202.938  mm,	Y = -249.725  mm,	Z = -231.016  mm,
	W = 0.000 deg,	P = 30.000 deg,	R = 179.752 deg
};
P[88]{
   GP1:
	UF : 0, UT : 1,		CONFIG : 'N U T, 0, 0, 0',
	X = 1202.947  mm,	Y = -247.725  mm,	Z = -230.999  mm,
	W = 0.000 deg,	P = 30.000 deg,	R = 179.752 deg
};
P[89]{
   GP1:
	UF : 0, UT : 1,		CONFIG : 'N U T, 0, 0, 0',
	X = 1202.956  mm,	Y = -245.725  mm,	Z = -230.983  mm,
	W = 0.000 deg,	P = 30.000 deg,	R = 179.752 deg
};
P[90]{
   GP1:
	UF : 0, UT : 1,		CONFIG : 'N U T, 0, 0, 0',
	X = 1202.965  mm,	Y = -243.725  mm,	Z = -230.966  mm,
	W = 0.000 deg,	P = 30.000 deg,	R = 179.752 deg
};
P[91]{
   GP1:
	UF : 0, UT : 1,		CONFIG : 'N U T, 0, 0, 0',
	X = 1202.973  mm,	Y = -241.725  mm,	Z = -230.949  mm,
	W = 0.000 deg,	P = 30.000 deg,	R = 179.752 deg
};
P[92]{
   GP1:
	UF : 0, UT : 1,		CONFIG : 'N U T, 0, 0, 0',
	X = 1202.982  mm,	Y = -239.725  mm,	Z = -230.932  mm,
	W = 0.000 deg,	P = 30.000 deg,	R = 179.752 deg
};
P[93]{
   GP1:
	UF : 0, UT : 1,		CONFIG : 'N U T, 0, 0, 0',
	X = 1202.991  mm,	Y = -237.725  mm,	Z = -230.916  mm,
	W = 0.000 deg,	P = 30.000 deg,	R = 179.752 deg
};
P[94]{
   GP1:
	UF : 0, UT : 1,		CONFIG : 'N U T, 0, 0, 0',
	X = 1202.999  mm,	Y = -235.725  mm,	Z = -230.899  mm,
	W = 0.000 deg,	P = 30.000 deg,	R = 179.752 deg
};
P[95]{
   GP1:
	UF : 0, UT : 1,		CONFIG : 'N U T, 0, 0, 0',
	X = 1203.008  mm,	Y = -233.726  mm,	Z = -230.882  mm,
	W = 0.000 deg,	P = 30.000 deg,	R = 179.752 deg
};
P[96]{
   GP1:
	UF : 0, UT : 1,		CONFIG : 'N U T, 0, 0, 0',
	X = 1203.017  mm,	Y = -231.726  mm,	Z = -230.865  mm,
	W = 0.000 deg,	P = 30.000 deg,	R = 179.752 deg
};
P[97]{
   GP1:
	UF : 0, UT : 1,		CONFIG : 'N U T, 0, 0, 0',
	X = 1203.025  mm,	Y = -229.726  mm,	Z = -230.848  mm,
	W = 0.000 deg,	P = 30.000 deg,	R = 179.752 deg
};
P[98]{
   GP1:
	UF : 0, UT : 1,		CONFIG : 'N U T, 0, 0, 0',
	X = 1203.034  mm,	Y = -227.726  mm,	Z = -230.832  mm,
	W = 0.000 deg,	P = 30.000 deg,	R = 179.752 deg
};
P[99]{
   GP1:
	UF : 0, UT : 1,		CONFIG : 'N U T, 0, 0, 0',
	X = 1203.043  mm,	Y = -225.726  mm,	Z = -230.815  mm,
	W = 0.000 deg,	P = 30.000 deg,	R = 179.752 deg
};
P[100]{
   GP1:
	UF : 0, UT : 1,		CONFIG : 'N U T, 0, 0, 0',
	X = 1203.051  mm,	Y = -223.726  mm,	Z = -230.798  mm,
	W = 0.000 deg,	P = 30.000 deg,	R = 179.752 deg
};
P[101]{
   GP1:
	UF : 0, UT : 1,		CONFIG : 'N U T, 0, 0, 0',
	X = 1203.060  mm,	Y = -221.726  mm,	Z = -230.781  mm,
	W = 0.000 deg,	P = 30.000 deg,	R = 179.752 deg
};
P[102]{
   GP1:
	UF : 0, UT : 1,		CONFIG : 'N U T, 0, 0, 0',
	X = 1203.069  mm,	Y = -219.726  mm,	Z = -230.765  mm,
	W = 0.000 deg,	P = 30.000 deg,	R = 179.752 deg
};
P[103]{
   GP1:
	UF : 0, UT : 1,		CONFIG : 'N U T, 0, 0, 0',
	X = 1203.077  mm,	Y = -217.726  mm,	Z = -230.748  mm,
	W = 0.000 deg,	P = 30.000 deg,	R = 179.752 deg
};
P[104]{
   GP1:
	UF : 0, UT : 1,		CONFIG : 'N U T, 0, 0, 0',
	X = 1203.086  mm,	Y = -215.726  mm,	Z = -230.731  mm,
	W = 0.000 deg,	P = 30.000 deg,	R = 179.752 deg
};
P[105]{
   GP1:
	UF : 0, UT : 1,		CONFIG : 'N U T, 0, 0, 0',
	X = 1203.095  mm,	Y = -213.726  mm,	Z = -230.714  mm,
	W = 0.000 deg,	P = 30.000 deg,	R = 179.752 deg
};
P[106]{
   GP1:
	UF : 0, UT : 1,		CONFIG : 'N U T, 0, 0, 0',
	X = 1203.103  mm,	Y = -211.726  mm,	Z = -230.698  mm,
	W = 0.000 deg,	P = 30.000 deg,	R = 179.752 deg
};
P[107]{
   GP1:
	UF : 0, UT : 1,		CONFIG : 'N U T, 0, 0, 0',
	X = 1203.112  mm,	Y = -209.727  mm,	Z = -230.681  mm,
	W = 0.000 deg,	P = 30.000 deg,	R = 179.752 deg
};
P[108]{
   GP1:
	UF : 0, UT : 1,		CONFIG : 'N U T, 0, 0, 0',
	X = 1203.121  mm,	Y = -207.727  mm,	Z = -230.664  mm,
	W = 0.000 deg,	P = 30.000 deg,	R = 179.752 deg
};
P[109]{
   GP1:
	UF : 0, UT : 1,		CONFIG : 'N U T, 0, 0, 0',
	X = 1203.129  mm,	Y = -205.727  mm,	Z = -230.647  mm,
	W = 0.000 deg,	P = 30.000 deg,	R = 172.310 deg
};
P[110]{
   GP1:
	UF : 0, UT : 1,		CONFIG : 'N U T, 0, 0, 0',
	X = 1203.138  mm,	Y = -203.727  mm,	Z = -230.630  mm,
	W = 0.000 deg,	P = 30.000 deg,	R = 168.360 deg
};
P[111]{
   GP1:
	UF : 0, UT : 1,		CONFIG : 'N U T, 0, 0, 0',
	X = 1203.147  mm,	Y = -201.727  mm,	Z = -230.614  mm,
	W = 0.000 deg,	P = 30.000 deg,	R = 164.410 deg
};
P[112]{
   GP1:
	UF : 0, UT : 1,		CONFIG : 'N U T, 0, 0, 0',
	X = 1203.155  mm,	Y = -199.727  mm,	Z = -230.597  mm,
	W = 0.000 deg,	P = 30.000 deg,	R = 160.459 deg
};
P[113]{
   GP1:
	UF : 0, UT : 1,		CONFIG : 'N U T, 0, 0, 0',
	X = 1203.162  mm,	Y = -198.274  mm,	Z = -230.585  mm,
	W = 0.000 deg,	P = 30.000 deg,	R = 160.000 deg
};
P[114]{
   GP1:
	UF : 0, UT : 1,		CONFIG : 'N U T, 0, 0, 0',
	X = 1203.516  mm,	Y = -197.865  mm,	Z = -230.661  mm,
	W = 0.000 deg,	P = 30.000 deg,	R = 160.000 deg
};
P[115]{
   GP1:
	UF : 0, UT : 1,		CONFIG : 'N U T, 0, 0, 0',
	X = 1204.813  mm,	Y = -196.368  mm,	Z = -230.942  mm,
	W = 0.000 deg,	P = 30.000 deg,	R = 160.000 deg
};
P[116]{
   GP1:
	UF : 0, UT : 1,		CONFIG : 'N U T, 0, 0, 0',
	X = 1206.109  mm,	Y = -194.871  mm,	Z = -231.223  mm,
	W = 0.000 deg,	P = 30.000 deg,	R = 160.000 deg
};
P[117]{
   GP1:
	UF : 0, UT : 1,		CONFIG : 'N U T, 0, 0, 0',
	X = 1207.406  mm,	Y = -193.374  mm,	Z = -231.503  mm,
	W = 0.000 deg,	P = 30.000 deg,	R = 160.000 deg
};
P[118]{
   GP1:
	UF : 0, UT : 1,		CONFIG : 'N U T, 0, 0, 0',
	X = 1208.702  mm,	Y = -191.878  mm,	Z = -231.784  mm,
	W = 0.000 deg,	P = 30.000 deg,	R = 160.000 deg
};
P[119]{
   GP1:
	UF : 0, UT : 1,		CONFIG : 'N U T, 0, 0, 0',
	X = 1209.999  mm,	Y = -190.381  mm,	Z = -232.065  mm,
	W = 0.000 deg,	P = 30.000 deg,	R = 160.000 deg
};
P[120]{
   GP1:
	UF : 0, UT : 1,		CONFIG : 'N U T, 0, 0, 0',
	X = 1211.295  mm,	Y = -188.884  mm,	Z = -232.345  mm,
	W = 0.000 deg,	P = 30.000 deg,	R = 160.000 deg
};
P[121]{
   GP1:
	UF : 0, UT : 1,		CONFIG : 'N U T, 0, 0, 0',
	X = 1212.592  mm,	Y = -187.387  mm,	Z = -232.626  mm,
	W = 0.000 deg,	P = 30.000 deg,	R = 160.000 deg
};
P[122]{
   GP1:
	UF : 0, UT : 1,		CONFIG : 'N U T, 0, 0, 0',
	X = 1213.888  mm,	Y = -185.891  mm,	Z = -232.907  mm,
	W = 0.000 deg,	P = 30.000 deg,	R = 160.000 deg
};
P[123]{
   GP1:
	UF : 0, UT : 1,		CONFIG : 'N U T, 0, 0, 0',
	X = 1215.185  mm,	Y = -184.394  mm,	Z = -233.187  mm,
	W = 0.000 deg,	P = 30.000 deg,	R = 160.000 deg
};
P[124]{
   GP1:
	UF : 0, UT : 1,		CONFIG : 'N U T, 0, 0, 0',
	X = 1216.481  mm,	Y = -182.897  mm,	Z = -233.468  mm,
	W = 0.000 deg,	P = 30.000 deg,	R = 160.000 deg
};
P[125]{
   GP1:
	UF : 0, UT : 1,		CONFIG : 'N U T, 0, 0, 0',
	X = 1217.778  mm,	Y = -181.400  mm,	Z = -233.749  mm,
	W = 0.000 deg,	P = 30.000 deg,	R = 160.000 deg
};
P[126]{
   GP1:
	UF : 0, UT : 1,		CONFIG : 'N U T, 0, 0, 0',
	X = 1219.074  mm,	Y = -179.903  mm,	Z = -234.029  mm,
	W = 0.000 deg,	P = 30.000 deg,	R = 160.000 deg
};
P[127]{
   GP1:
	UF : 0, UT : 1,		CONFIG : 'N U T, 0, 0, 0',
	X = 1220.371  mm,	Y = -178.407  mm,	Z = -234.310  mm,
	W = 0.000 deg,	P = 30.000 deg,	R = 160.000 deg
};
P[128]{
   GP1:
	UF : 0, UT : 1,		CONFIG : 'N U T, 0, 0, 0',
	X = 1221.667  mm,	Y = -176.910  mm,	Z = -234.591  mm,
	W = 0.000 deg,	P = 30.000 deg,	R = 160.000 deg
};
P[129]{
   GP1:
	UF : 0, UT : 1,		CONFIG : 'N U T, 0, 0, 0',
	X = 1222.964  mm,	Y = -175.413  mm,	Z = -234.871  mm,
	W = 0.000 deg,	P = 30.000 deg,	R = 160.000 deg
};
P[130]{
   GP1:
	UF : 0, UT : 1,		CONFIG : 'N U T, 0, 0, 0',
	X = 1224.260  mm,	Y = -173.916  mm,	Z = -235.152  mm,
	W = 0.000 deg,	P = 30.000 deg,	R = 160.000 deg
};
P[131]{
   GP1:
	UF : 0, UT : 1,		CONFIG : 'N U T, 0, 0, 0',
	X = 1225.557  mm,	Y = -172.420  mm,	Z = -235.433  mm,
	W = 0.000 deg,	P = 30.000 deg,	R = 160.000 deg
};
P[132]{
   GP1:
	UF : 0, UT : 1,		CONFIG : 'N U T, 0, 0, 0',
	X = 1226.853  mm,	Y = -170.923  mm,	Z = -235.713  mm,
	W = 0.000 deg,	P = 30.000 deg,	R = 160.000 deg
};
P[133]{
   GP1:
	UF : 0, UT : 1,		CONFIG : 'N U T, 0, 0, 0',
	X = 1228.150  mm,	Y = -169.426  mm,	Z = -235.994  mm,
	W = 0.000 deg,	P = 30.000 deg,	R = 160.000 deg
};
P[134]{
   GP1:
	UF : 0, UT : 1,		CONFIG : 'N U T, 0, 0, 0',
	X = 1229.446  mm,	Y = -167.929  mm,	Z = -236.275  mm,
	W = 0.000 deg,	P = 30.000 deg,	R = 161.238 deg
};
P[135]{
   GP1:
	UF : 0, UT : 1,		CONFIG : 'N U T, 0, 0, 0',
	X = 1230.743  mm,	Y = -166.432  mm,	Z = -236.555  mm,
	W = 0.000 deg,	P = 30.000 deg,	R = 165.761 deg
};
P[136]{
   GP1:
	UF : 0, UT : 1,		CONFIG : 'N U T, 0, 0, 0',
	X = 1232.039  mm,	Y = -164.936  mm,	Z = -236.836  mm,
	W = 0.000 deg,	P = 30.000 deg,	R = 170.284 deg
};
P[137]{
   GP1:
	UF : 0, UT : 1,		CONFIG : 'N U T, 0, 0, 0',
	X = 1233.336  mm,	Y = -163.439  mm,	Z = -237.117  mm,
	W = 0.000 deg,	P = 30.000 deg,	R = 174.808 deg
};
P[138]{
   GP1:
	UF : 0, UT : 1,		CONFIG : 'N U T, 0, 0, 0',
	X = 1234.632  mm,	Y = -161.942  mm,	Z = -237.397  mm,
	W = 0.000 deg,	P = 30.000 deg,	R = 179.331 deg
};
P[139]{
   GP1:
	UF : 0, UT : 1,		CONFIG : 'N U T, 0, 0, 0',
	X = 1235.891  mm,	Y = -160.489  mm,	Z = -237.670  mm,
	W = 0.000 deg,	P = 30.000 deg,	R = -177.384 deg
};
P[140]{
   GP1:
	UF : 0, UT : 1,		CONFIG : 'N U T, 0, 0, 0',
	X = 1235.889  mm,	Y = -160.431  mm,	Z = -237.669  mm,
	W = 0.000 deg,	P = 30.000 deg,	R = -177.384 deg
};
P[141]{
   GP1:
	UF : 0, UT : 1,		CONFIG : 'N U T, 0, 0, 0',
	X = 1235.797  mm,	Y = -158.434  mm,	Z = -237.616  mm,
	W = 0.000 deg,	P = 30.000 deg,	R = -177.384 deg
};
P[142]{
   GP1:
	UF : 0, UT : 1,		CONFIG : 'N U T, 0, 0, 0',
	X = 1235.706  mm,	Y = -156.436  mm,	Z = -237.563  mm,
	W = 0.000 deg,	P = 30.000 deg,	R = -177.384 deg
};
P[143]{
   GP1:
	UF : 0, UT : 1,		CONFIG : 'N U T, 0, 0, 0',
	X = 1235.615  mm,	Y = -154.439  mm,	Z = -237.510  mm,
	W = 0.000 deg,	P = 30.000 deg,	R = -177.384 deg
};
P[144]{
   GP1:
	UF : 0, UT : 1,		CONFIG : 'N U T, 0, 0, 0',
	X = 1235.524  mm,	Y = -152.442  mm,	Z = -237.457  mm,
	W = 0.000 deg,	P = 30.000 deg,	R = -177.384 deg
};
P[145]{
   GP1:
	UF : 0, UT : 1,		CONFIG : 'N U T, 0, 0, 0',
	X = 1235.432  mm,	Y = -150.445  mm,	Z = -237.404  mm,
	W = 0.000 deg,	P = 30.000 deg,	R = -177.384 deg
};
P[146]{
   GP1:
	UF : 0, UT : 1,		CONFIG : 'N U T, 0, 0, 0',
	X = 1235.341  mm,	Y = -148.448  mm,	Z = -237.351  mm,
	W = 0.000 deg,	P = 30.000 deg,	R = -177.384 deg
};
P[147]{
   GP1:
	UF : 0, UT : 1,		CONFIG : 'N U T, 0, 0, 0',
	X = 1235.250  mm,	Y = -146.450  mm,	Z = -237.299  mm,
	W = 0.000 deg,	P = 30.000 deg,	R = -177.384 deg
};
P[148]{
   GP1:
	UF : 0, UT : 1,		CONFIG : 'N U T, 0, 0, 0',
	X = 1235.158  mm,	Y = -144.453  mm,	Z = -237.246  mm,
	W = 0.000 deg,	P = 30.000 deg,	R = -177.384 deg
};
P[149]{
   GP1:
	UF : 0, UT : 1,		CONFIG : 'N U T, 0, 0, 0',
	X = 1235.067  mm,	Y = -142.456  mm,	Z = -237.193  mm,
	W = 0.000 deg,	P = 30.000 deg,	R = -177.384 deg
};
P[150]{
   GP1:
	UF : 0, UT : 1,		CONFIG : 'N U T, 0, 0, 0',
	X = 1234.976  mm,	Y = -140.459  mm,	Z = -237.140  mm,
	W = 0.000 deg,	P = 30.000 deg,	R = -177.384 deg
};
P[151]{
   GP1:
	UF : 0, UT : 1,		CONFIG : 'N U T, 0, 0, 0',
	X = 1234.885  mm,	Y = -138.461  mm,	Z = -237.087  mm,
	W = 0.000 deg,	P = 30.000 deg,	R = -177.384 deg
};
P[152]{
   GP1:
	UF : 0, UT : 1,		CONFIG : 'N U T, 0, 0, 0',
	X = 1234.793  mm,	Y = -136.464  mm,	Z = -237.034  mm,
	W = 0.000 deg,	P = 30.000 deg,	R = -177.384 deg
};
P[153]{
   GP1:
	UF : 0, UT : 1,		CONFIG : 'N U T, 0, 0, 0',
	X = 1234.702  mm,	Y = -134.467  mm,	Z = -236.981  mm,
	W = 0.000 deg,	P = 30.000 deg,	R = -177.384 deg
};
P[154]{
   GP1:
	UF : 0, UT : 1,		CONFIG : 'N U T, 0, 0, 0',
	X = 1234.611  mm,	Y = -132.470  mm,	Z = -236.929  mm,
	W = 0.000 deg,	P = 30.000 deg,	R = -177.384 deg
};
P[155]{
   GP1:
	UF : 0, UT : 1,		CONFIG : 'N U T, 0, 0, 0',
	X = 1234.520  mm,	Y = -130.473  mm,	Z = -236.876  mm,
	W = 0.000 deg,	P = 30.000 deg,	R = -177.384 deg
};
P[156]{
   GP1:
	UF : 0, UT : 1,		CONFIG : 'N U T, 0, 0, 0',
	X = 1234.428  mm,	Y = -128.475  mm,	Z = -236.823  mm,
	W = 0.000 deg,	P = 30.000 deg,	R = -177.384 deg
};
P[157]{
   GP1:
	UF : 0, UT : 1,		CONFIG : 'N U T, 0, 0, 0',
	X = 1234.337  mm,	Y = -126.478  mm,	Z = -236.770  mm,
	W = 0.000 deg,	P = 30.000 deg,	R = -177.384 deg
};
P[158]{
   GP1:
	UF : 0, UT : 1,		CONFIG : 'N U T, 0, 0, 0',
	X = 1234.246  mm,	Y = -124.481  mm,	Z = -236.717  mm,
	W = 0.000 deg,	P = 30.000 deg,	R = -177.384 deg
};
P[159]{
   GP1:
	UF : 0, UT : 1,		CONFIG : 'N U T, 0, 0, 0',
	X = 1234.155  mm,	Y = -122.484  mm,	Z = -236.664  mm,
	W = 0.000 deg,	P = 30.000 deg,	R = -177.384 deg
};
P[160]{
   GP1:
	UF : 0, UT : 1,		CONFIG : 'N U T, 0, 0, 0',
	X = 1234.063  mm,	Y = -120.487  mm,	Z = -236.611  mm,
	W = 0.000 deg,	P = 30.000 deg,	R = -177.384 deg
};
P[161]{
   GP1:
	UF : 0, UT : 1,		CONFIG : 'N U T, 0, 0, 0',
	X = 1233.972  mm,	Y = -118.489  mm,	Z = -236.559  mm,
	W = 0.000 deg,	P = 30.000 deg,	R = -177.384 deg
};
P[162]{
   GP1:
	UF : 0, UT : 1,		CONFIG : 'N U T, 0, 0, 0',
	X = 1233.881  mm,	Y = -116.492  mm,	Z = -236.506  mm,
	W = 0.000 deg,	P = 30.000 deg,	R = -177.384 deg
};
P[163]{
   GP1:
	UF : 0, UT : 1,		CONFIG : 'N U T, 0, 0, 0',
	X = 1233.790  mm,	Y = -114.495  mm,	Z = -236.453  mm,
	W = 0.000 deg,	P = 30.000 deg,	R = -177.384 deg
};
P[164]{
   GP1:
	UF : 0, UT : 1,		CONFIG : 'N U T, 0, 0, 0',
	X = 1233.698  mm,	Y = -112.498  mm,	Z = -236.400  mm,
	W = 0.000 deg,	P = 30.000 deg,	R = -173.807 deg
};
P[165]{
   GP1:
	UF : 0, UT : 1,		CONFIG : 'N U T, 0, 0, 0',
	X = 1233.607  mm,	Y = -110.500  mm,	Z = -236.347  mm,
	W = 0.000 deg,	P = 30.000 deg,	R = -170.330 deg
};
P[166]{
   GP1:
	UF : 0, UT : 1,		CONFIG : 'N U T, 0, 0, 0',
	X = 1233.516  mm,	Y = -108.503  mm,	Z = -236.294  mm,
	W = 0.000 deg,	P = 30.000 deg,	R = -166.853 deg
};
P[167]{
   GP1:
	UF : 0, UT : 1,		CONFIG : 'N U T, 0, 0, 0',
	X = 1233.425  mm,	Y = -106.506  mm,	Z = -236.241  mm,
	W = 0.000 deg,	P = 30.000 deg,	R = -163.376 deg
};
P[168]{
   GP1:
	UF : 0, UT : 1,		CONFIG : 'N U T, 0, 0, 0',
	X = 1233.333  mm,	Y = -104.509  mm,	Z = -236.189  mm,
	W = 0.000 deg,	P = 30.000 deg,	R = -160.000 deg
};
P[169]{
   GP1:
	UF : 0, UT : 1,		CONFIG : 'N U T, 0, 0, 0',
	X = 1233.296  mm,	Y = -103.684  mm,	Z = -236.167  mm,
	W = 0.000 deg,	P = 30.000 deg,	R = -160.000 deg
};
P[170]{
   GP1:
	UF : 0, UT : 1,		CONFIG : 'N U T, 0, 0, 0',
	X = 1232.479  mm,	Y = -102.862  mm,	Z = -235.977  mm,
	W = 0.000 deg,	P = 30.000 deg,	R = -160.000 deg
};
P[171]{
   GP1:
	UF : 0, UT : 1,		CONFIG : 'N U T, 0, 0, 0',
	X = 1231.088  mm,	Y = -101.462  mm,	Z = -235.653  mm,
	W = 0.000 deg,	P = 30.000 deg,	R = -160.000 deg
};
P[172]{
   GP1:
	UF : 0, UT : 1,		CONFIG : 'N U T, 0, 0, 0',
	X = 1229.697  mm,	Y = -100.062  mm,	Z = -235.329  mm,
	W = 0.000 deg,	P = 30.000 deg,	R = -160.000 deg
};
P[173]{
   GP1:
	UF : 0, UT : 1,		CONFIG : 'N U T, 0, 0, 0',
	X = 1228.306  mm,	Y = -98.662  mm,	Z = -235.006  mm,
	W = 0.000 deg,	P = 30.000 deg,	R = -160.000 deg
};
P[174]{
   GP1:
	UF : 0, UT : 1,		CONFIG : 'N U T, 0, 0, 0',
	X = 1226.915  mm,	Y = -97.262  mm,	Z = -234.682  mm,
	W = 0.000 deg,	P = 30.000 deg,	R = -160.000 deg
};
P[175]{
   GP1:
	UF : 0, UT : 1,		CONFIG : 'N U T, 0, 0, 0',
	X = 1225.524  mm,	Y = -95.861  mm,	Z = -234.358  mm,
	W = 0.000 deg,	P = 30.000 deg,	R = -160.000 deg
};
P[176]{
   GP1:
	UF : 0, UT : 1,		CONFIG : 'N U T, 0, 0, 0',
	X = 1224.133  mm,	Y = -94.461  mm,	Z = -234.035  mm,
	W = 0.000 deg,	P = 30.000 deg,	R = -160.000 deg
};
P[177]{
   GP1:
	UF : 0, UT : 1,		CONFIG : 'N U T, 0, 0, 0',
	X = 1222.742  mm,	Y = -93.061  mm,	Z = -233.711  mm,
	W = 0.000 deg,	P = 30.000 deg,	R = -160.000 deg
};
P[178]{
   GP1:
	UF : 0, UT : 1,		CONFIG : 'N U T, 0, 0, 0',
	X = 1221.351  mm,	Y = -91.661  mm,	Z = -233.387  mm,
	W = 0.000 deg,	P = 30.000 deg,	R = -160.000 deg
};
P[179]{
   GP1:
	UF : 0, UT : 1,		CONFIG : 'N U T, 0, 0, 0',
	X = 1219.960  mm,	Y = -90.261  mm,	Z = -233.064  mm,
	W = 0.000 deg,	P = 30.000 deg,	R = -160.000 deg
};
P[180]{
   GP1:
	UF : 0, UT : 1,		CONFIG : 'N U T, 0, 0, 0',
	X = 1218.569  mm,	Y = -88.861  mm,	Z = -232.740  mm,
	W = 0.000 deg,	P = 30.000 deg,	R = -160.000 deg
};
P[181]{
   GP1:
	UF : 0, UT : 1,		CONFIG : 'N U T, 0, 0, 0',
	X = 1217.178  mm,	Y = -87.460  mm,	Z = -232.416  mm,
	W = 0.000 deg,	P = 30.000 deg,	R = -160.000 deg
};
P[182]{
   GP1:
	UF : 0, UT : 1,		CONFIG : 'N U T, 0, 0, 0',
	X = 1215.787  mm,	Y = -86.060  mm,	Z = -232.093  mm,
	W = 0.000 deg,	P = 30.000 deg,	R = -160.000 deg
};
P[183]{
   GP1:
	UF : 0, UT : 1,		CONFIG : 'N U T, 0, 0, 0',
	X = 1214.396  mm,	Y = -84.660  mm,	Z = -231.769  mm,
	W = 0.000 deg,	P = 30.000 deg,	R = -160.000 deg
};
P[184]{
   GP1:
	UF : 0, UT : 1,		CONFIG : 'N U T, 0, 0, 0',
	X = 1213.005  mm,	Y = -83.260  mm,	Z = -231.445  mm,
	W = 0.000 deg,	P = 30.000 deg,	R = -160.000 deg
};
P[185]{
   GP1:
	UF : 0, UT : 1,		CONFIG : 'N U T, 0, 0, 0',
	X = 1211.614  mm,	Y = -81.860  mm,	Z = -231.121  mm,
	W = 0.000 deg,	P = 30.000 deg,	R = -160.000 deg
};
P[186]{
   GP1:
	UF : 0, UT : 1,		CONFIG : 'N U T, 0, 0, 0',
	X = 1210.223  mm,	Y = -80.460  mm,	Z = -230.798  mm,
	W = 0.000 deg,	P = 30.000 deg,	R = -160.000 deg
};
P[187]{
   GP1:
	UF : 0, UT : 1,		CONFIG : 'N U T, 0, 0, 0',
	X = 1208.832  mm,	Y = -79.060  mm,	Z = -230.474  mm,
	W = 0.000 deg,	P = 30.000 deg,	R = -160.000 deg
};
P[188]{
   GP1:
	UF : 0, UT : 1,		CONFIG : 'N U T, 0, 0, 0',
	X = 1207.441  mm,	Y = -77.659  mm,	Z = -230.150  mm,
	W = 0.000 deg,	P = 30.000 deg,	R = -160.000 deg
};
P[189]{
   GP1:
	UF : 0, UT : 1,		CONFIG : 'N U T, 0, 0, 0',
	X = 1206.050  mm,	Y = -76.259  mm,	Z = -229.827  mm,
	W = 0.000 deg,	P = 30.000 deg,	R = -160.000 deg
};
P[190]{
   GP1:
	UF : 0, UT : 1,		CONFIG : 'N U T, 0, 0, 0',
	X = 1204.660  mm,	Y = -74.859  mm,	Z = -229.503  mm,
	W = 0.000 deg,	P = 30.000 deg,	R = -160.000 deg
};
P[191]{
   GP1:
	UF : 0, UT : 1,		CONFIG : 'N U T, 0, 0, 0',
	X = 1203.269  mm,	Y = -73.459  mm,	Z = -229.179  mm,
	W = 0.000 deg,	P = 30.000 deg,	R = -166.498 deg
};
P[192]{
   GP1:
	UF : 0, UT : 1,		CONFIG : 'N U T, 0, 0, 0',
	X = 1201.878  mm,	Y = -72.059  mm,	Z = -228.856  mm,
	W = 0.000 deg,	P = 30.000 deg,	R = -170.593 deg
};
P[193]{
   GP1:
	UF : 0, UT : 1,		CONFIG : 'N U T, 0, 0, 0',
	X = 1200.487  mm,	Y = -70.659  mm,	Z = -228.532  mm,
	W = 0.000 deg,	P = 30.000 deg,	R = -174.687 deg
};
P[194]{
   GP1:
	UF : 0, UT : 1,		CONFIG : 'N U T, 0, 0, 0',
	X = 1199.096  mm,	Y = -69.258  mm,	Z = -228.208  mm,
	W = 0.000 deg,	P = 30.000 deg,	R = -178.782 deg
};
P[195]{
   GP1:
	UF : 0, UT : 1,		CONFIG : 'N U T, 0, 0, 0',
	X = 1197.705  mm,	Y = -67.858  mm,	Z = -227.885  mm,
	W = 0.000 deg,	P = 30.000 deg,	R = 179.528 deg
};
P[196]{
   GP1:
	UF : 0, UT : 1,		CONFIG : 'N U T, 0, 0, 0',
	X = 1197.676  mm,	Y = -67.829  mm,	Z = -227.878  mm,
	W = 0.000 deg,	P = 30.000 deg,	R = 179.528 deg
};
P[197]{
   GP1:
	UF : 0, UT : 1,		CONFIG : 'N U T, 0, 0, 0',
	X = 1197.692  mm,	Y = -65.871  mm,	Z = -227.859  mm,
	W = 0.000 deg,	P = 30.000 deg,	R = 179.528 deg
};
P[198]{
   GP1:
	UF : 0, UT : 1,		CONFIG : 'N U T, 0, 0, 0',
	X = 1197.708  mm,	Y = -63.871  mm,	Z = -227.841  mm,
	W = 0.000 deg,	P = 30.000 deg,	R = 179.528 deg
};
P[199]{
   GP1:
	UF : 0, UT : 1,		CONFIG : 'N U T, 0, 0, 0',
	X = 1197.725  mm,	Y = -61.871  mm,	Z = -227.822  mm,
	W = 0.000 deg,	P = 30.000 deg,	R = 179.528 deg
};
P[200]{
   GP1:
	UF : 0, UT : 1,		CONFIG : 'N U T, 0, 0, 0',
	X = 1197.741  mm,	Y = -59.871  mm,	Z = -227.803  mm,
	W = 0.000 deg,	P = 30.000 deg,	R = 179.528 deg
};
P[201]{
   GP1:
	UF : 0, UT : 1,		CONFIG : 'N U T, 0, 0, 0',
	X = 1197.758  mm,	Y = -57.872  mm,	Z = -227.784  mm,
	W = 0.000 deg,	P = 30.000 deg,	R = 179.528 deg
};
P[202]{
   GP1:
	UF : 0, UT : 1,		CONFIG : 'N U T, 0, 0, 0',
	X = 1197.774  mm,	Y = -55.872  mm,	Z = -227.765  mm,
	W = 0.000 deg,	P = 30.000 deg,	R = 179.528 deg
};
P[203]{
   GP1:
	UF : 0, UT : 1,		CONFIG : 'N U T, 0, 0, 0',
	X = 1197.791  mm,	Y = -53.872  mm,	Z = -227.746  mm,
	W = 0.000 deg,	P = 30.000 deg,	R = 179.528 deg
};
P[204]{
   GP1:
	UF : 0, UT : 1,		CONFIG : 'N U T, 0, 0, 0',
	X = 1197.807  mm,	Y = -51.872  mm,	Z = -227.727  mm,
	W = 0.000 deg,	P = 30.000 deg,	R = 179.528 deg
};
P[205]{
   GP1:
	UF : 0, UT : 1,		CONFIG : 'N U T, 0, 0, 0',
	X = 1197.824  mm,	Y = -49.872  mm,	Z = -227.708  mm,
	W = 0.000 deg,	P = 30.000 deg,	R = 179.528 deg
};
P[206]{
   GP1:
	UF : 0, UT : 1,		CONFIG : 'N U T, 0, 0, 0',
	X = 1197.840  mm,	Y = -47.872  mm,	Z = -227.689  mm,
	W = 0.000 deg,	P = 30.000 deg,	R = 179.528 deg
};
P[207]{
   GP1:
	UF : 0, UT : 1,		CONFIG : 'N U T, 0, 0, 0',
	X = 1197.857  mm,	Y = -45.872  mm,	Z = -227.670  mm,
	W = 0.000 deg,	P = 30.000 deg,	R = 179.528 deg
};
P[208]{
   GP1:
	UF : 0, UT : 1,		CONFIG : 'N U T, 0, 0, 0',
	X = 1197.873  mm,	Y = -43.873  mm,	Z = -227.651  mm,
	W = 0.000 deg,	P = 30.000 deg,	R = 179.528 deg
};
P[209]{
   GP1:
	UF : 0, UT : 1,		CONFIG : 'N U T, 0, 0, 0',
	X = 1197.890  mm,	Y = -41.873  mm,	Z = -227.633  mm,
	W = 0.000 deg,	P = 30.000 deg,	R = 179.528 deg
};
P[210]{
   GP1:
	UF : 0, UT : 1,		CONFIG : 'N U T, 0, 0, 0',
	X = 1197.906  mm,	Y = -39.873  mm,	Z = -227.614  mm,
	W = 0.000 deg,	P = 30.000 deg,	R = 179.528 deg
};
P[211]{
   GP1:
	UF : 0, UT : 1,		CONFIG : 'N U T, 0, 0, 0',
	X = 1197.923  mm,	Y = -37.873  mm,	Z = -227.595  mm,
	W = 0.000 deg,	P = 30.000 deg,	R = 179.528 deg
};
P[212]{
   GP1:
	UF : 0, UT : 1,		CONFIG : 'N U T, 0, 0, 0',
	X = 1197.939  mm,	Y = -35.873  mm,	Z = -227.576  mm,
	W = 0.000 deg,	P = 30.000 deg,	R = 179.528 deg
};
P[213]{
   GP1:
	UF : 0, UT : 1,		CONFIG : 'N U T, 0, 0, 0',
	X = 1197.956  mm,	Y = -33.873  mm,	Z = -227.557  mm,
	W = 0.000 deg,	P = 30.000 deg,	R = 179.528 deg
};
P[214]{
   GP1:
	UF : 0, UT : 1,		CONFIG : 'N U T, 0, 0, 0',
	X = 1197.972  mm,	Y = -31.874  mm,	Z = -227.538  mm,
	W = 0.000 deg,	P = 30.000 deg,	R = 179.528 deg
};
P[215]{
   GP1:
	UF : 0, UT : 1,		CONFIG : 'N U T, 0, 0, 0',
	X = 1197.989  mm,	Y = -29.874  mm,	Z = -227.519  mm,
	W = 0.000 deg,	P = 30.000 deg,	R = 179.528 deg
};
P[216]{
   GP1:
	UF : 0, UT : 1,		CONFIG : 'N U T, 0, 0, 0',
	X = 1198.005  mm,	Y = -27.874  mm,	Z = -227.500  mm,
	W = 0.000 deg,	P = 30.000 deg,	R = 179.528 deg
};
P[217]{
   GP1:
	UF : 0, UT : 1,		CONFIG : 'N U T, 0, 0, 0',
	X = 1198.021  mm,	Y = -25.874  mm,	Z = -227.481  mm,
	W = 0.000 deg,	P = 30.000 deg,	R = 179.528 deg
};
P[218]{
   GP1:
	UF : 0, UT : 1,		CONFIG : 'N U T, 0, 0, 0',
	X = 1198.038  mm,	Y = -23.874  mm,	Z = -227.462  mm,
	W = 0.000 deg,	P = 30.000 deg,	R = 179.528 deg
};
P[219]{
   GP1:
	UF : 0, UT : 1,		CONFIG : 'N U T, 0, 0, 0',
	X = 1198.054  mm,	Y = -21.874  mm,	Z = -227.443  mm,
	W = 0.000 deg,	P = 30.000 deg,	R = 179.528 deg
};
P[220]{
   GP1:
	UF : 0, UT : 1,		CONFIG : 'N U T, 0, 0, 0',
	X = 1198.071  mm,	Y = -19.875  mm,	Z = -227.424  mm,
	W = 0.000 deg,	P = 30.000 deg,	R = 175.703 deg
};
P[221]{
   GP1:
	UF : 0, UT : 1,		CONFIG : 'N U T, 0, 0, 0',
	X = 1198.087  mm,	Y = -17.875  mm,	Z = -227.406  mm,
	W = 0.000 deg,	P = 30.000 deg,	R = 171.798 deg
};
P[222]{
   GP1:
	UF : 0, UT : 1,		CONFIG : 'N U T, 0, 0, 0',
	X = 1198.104  mm,	Y = -15.875  mm,	Z = -227.387  mm,
	W = 0.000 deg,	P = 30.000 deg,	R = 167.892 deg
};
P[223]{
   GP1:
	UF : 0, UT : 1,		CONFIG : 'N U T, 0, 0, 0',
	X = 1198.120  mm,	Y = -13.875  mm,	Z = -227.368  mm,
	W = 0.000 deg,	P = 30.000 deg,	R = 163.987 deg
};
P[224]{
   GP1:
	UF : 0, UT : 1,		CONFIG : 'N U T, 0, 0, 0',
	X = 1198.137  mm,	Y = -11.875  mm,	Z = -227.349  mm,
	W = 0.000 deg,	P = 30.000 deg,	R = 160.081 deg
};
P[225]{
   GP1:
	UF : 0, UT : 1,		CONFIG : 'N U T, 0, 0, 0',
	X = 1198.153  mm,	Y = -9.875  mm,	Z = -227.330  mm,
	W = 0.000 deg,	P = 30.000 deg,	R = 160.000 deg
};
P[226]{
   GP1:
	UF : 0, UT : 1,		CONFIG : 'N U T, 0, 0, 0',
	X = 1198.154  mm,	Y = -9.843  mm,	Z = -227.330  mm,
	W = 0.000 deg,	P = 30.000 deg,	R = 160.000 deg
};
P[227]{
   GP1:
	UF : 0, UT : 1,		CONFIG : 'N U T, 0, 0, 0',
	X = 1199.459  mm,	Y = -8.400  mm,	Z = -227.624  mm,
	W = 0.000 deg,	P = 30.000 deg,	R = 160.000 deg
};
P[228]{
   GP1:
	UF : 0, UT : 1,		CONFIG : 'N U T, 0, 0, 0',
	X = 1200.785  mm,	Y = -6.933  mm,	Z = -227.923  mm,
	W = 0.000 deg,	P = 30.000 deg,	R = 160.000 deg
};
P[229]{
   GP1:
	UF : 0, UT : 1,		CONFIG : 'N U T, 0, 0, 0',
	X = 1202.111  mm,	Y = -5.466  mm,	Z = -228.222  mm,
	W = 0.000 deg,	P = 30.000 deg,	R = 160.000 deg
};
P[230]{
   GP1:
	UF : 0, UT : 1,		CONFIG : 'N U T, 0, 0, 0',
	X = 1203.437  mm,	Y = -3.999  mm,	Z = -228.521  mm,
	W = 0.000 deg,	P = 30.000 deg,	R = 160.000 deg
};
P[231]{
   GP1:
	UF : 0, UT : 1,		CONFIG : 'N U T, 0, 0, 0',
	X = 1204.763  mm,	Y = -2.532  mm,	Z = -228.821  mm,
	W = 0.000 deg,	P = 30.000 deg,	R = 160.000 deg
};
P[232]{
   GP1:
	UF : 0, UT : 1,		CONFIG : 'N U T, 0, 0, 0',
	X = 1206.089  mm,	Y = -1.066  mm,	Z = -229.120  mm,
	W = 0.000 deg,	P = 30.000 deg,	R = 160.000 deg
};
P[233]{
   GP1:
	UF : 0, UT : 1,		CONFIG : 'N U T, 0, 0, 0',
	X = 1207.416  mm,	Y = 0.401  mm,	Z = -229.419  mm,
	W = 0.000 deg,	P = 30.000 deg,	R = 160.000 deg
};
P[234]{
   GP1:
	UF : 0, UT : 1,		CONFIG : 'N U T, 0, 0, 0',
	X = 1208.742  mm,	Y = 1.868  mm,	Z = -229.718  mm,
	W = 0.000 deg,	P = 30.000 deg,	R = 160.000 deg
};
P[235]{
   GP1:
	UF : 0, UT : 1,		CONFIG : 'N U T, 0, 0, 0',
	X = 1210.068  mm,	Y = 3.335  mm,	Z = -230.017  mm,
	W = 0.000 deg,	P = 30.000 deg,	R = 160.000 deg
};
P[236]{
   GP1:
	UF : 0, UT : 1,		CONFIG : 'N U T, 0, 0, 0',
	X = 1211.394  mm,	Y = 4.802  mm,	Z = -230.316  mm,
	W = 0.000 deg,	P = 30.000 deg,	R = 160.000 deg
};
P[237]{
   GP1:
	UF : 0, UT : 1,		CONFIG : 'N U T, 0, 0, 0',
	X = 1212.720  mm,	Y = 6.269  mm,	Z = -230.616  mm,
	W = 0.000 deg,	P = 30.000 deg,	R = 160.000 deg
};
P[238]{
   GP1:
	UF : 0, UT : 1,		CONFIG : 'N U T, 0, 0, 0',
	X = 1214.047  mm,	Y = 7.736  mm,	Z = -230.915  mm,
	W = 0.000 deg,	P = 30.000 deg,	R = 160.000 deg
};
P[239]{
   GP1:
	UF : 0, UT : 1,		CONFIG : 'N U T, 0, 0, 0',
	X = 1215.373  mm,	Y = 9.203  mm,	Z = -231.214  mm,
	W = 0.000 deg,	P = 30.000 deg,	R = 160.000 deg
};
P[240]{
   GP1:
	UF : 0, UT : 1,		CONFIG : 'N U T, 0, 0, 0',
	X = 1216.699  mm,	Y = 10.670  mm,	Z = -231.513  mm,
	W = 0.000 deg,	P = 30.000 deg,	R = 160.000 deg
};
P[241]{
   GP1:
	UF : 0, UT : 1,		CONFIG : 'N U T, 0, 0, 0',
	X = 1218.025  mm,	Y = 12.136  mm,	Z = -231.812  mm,
	W = 0.000 deg,	P = 30.000 deg,	R = 160.000 deg
};
P[242]{
   GP1:
	UF : 0, UT : 1,		CONFIG : 'N U T, 0, 0, 0',
	X = 1219.351  mm,	Y = 13.603  mm,	Z = -232.111  mm,
	W = 0.000 deg,	P = 30.000 deg,	R = 160.000 deg
};
P[243]{
   GP1:
	UF : 0, UT : 1,		CONFIG : 'N U T, 0, 0, 0',
	X = 1220.677  mm,	Y = 15.070  mm,	Z = -232.411  mm,
	W = 0.000 deg,	P = 30.000 deg,	R = 160.000 deg
};
P[244]{
   GP1:
	UF : 0, UT : 1,		CONFIG : 'N U T, 0, 0, 0',
	X = 1222.004  mm,	Y = 16.537  mm,	Z = -232.710  mm,
	W = 0.000 deg,	P = 30.000 deg,	R = 160.000 deg
};
P[245]{
   GP1:
	UF : 0, UT : 1,		CONFIG : 'N U T, 0, 0, 0',
	X = 1223.330  mm,	Y = 18.004  mm,	Z = -233.009  mm,
	W = 0.000 deg,	P = 30.000 deg,	R = 160.000 deg
};
P[246]{
   GP1:
	UF : 0, UT : 1,		CONFIG : 'N U T, 0, 0, 0',
	X = 1224.656  mm,	Y = 19.471  mm,	Z = -233.308  mm,
	W = 0.000 deg,	P = 30.000 deg,	R = 160.000 deg
};
P[247]{
   GP1:
	UF : 0, UT : 1,		CONFIG : 'N U T, 0, 0, 0',
	X = 1225.982  mm,	Y = 20.938  mm,	Z = -233.607  mm,
	W = 0.000 deg,	P = 30.000 deg,	R = 160.000 deg
};
P[248]{
   GP1:
	UF : 0, UT : 1,		CONFIG : 'N U T, 0, 0, 0',
	X = 1227.308  mm,	Y = 22.405  mm,	Z = -233.906  mm,
	W = 0.000 deg,	P = 30.000 deg,	R = 168.857 deg
};
P[249]{
   GP1:
	UF : 0, UT : 1,		CONFIG : 'N U T, 0, 0, 0',
	X = 1228.635  mm,	Y = 23.872  mm,	Z = -234.205  mm,
	W = 0.000 deg,	P = 30.000 deg,	R = 173.321 deg
};
P[250]{
   GP1:
	UF : 0, UT : 1,		CONFIG : 'N U T, 0, 0, 0',
	X = 1229.961  mm,	Y = 25.338  mm,	Z = -234.505  mm,
	W = 0.000 deg,	P = 30.000 deg,	R = 177.786 deg
};
P[251]{
   GP1:
	UF : 0, UT : 1,		CONFIG : 'N U T, 0, 0, 0',
	X = 1231.287  mm,	Y = 26.805  mm,	Z = -234.804  mm,
	W = 0.000 deg,	P = 30.000 deg,	R = -177.750 deg
};
P[252]{
   GP1:
	UF : 0, UT : 1,		CONFIG : 'N U T, 0, 0, 0',
	X = 1232.414  mm,	Y = 28.052  mm,	Z = -235.058  mm,
	W = 0.000 deg,	P = 30.000 deg,	R = -177.679 deg
};
P[253]{
   GP1:
	UF : 0, UT : 1,		CONFIG : 'N U T, 0, 0, 0',
	X = 1232.402  mm,	Y = 28.352  mm,	Z = -235.053  mm,
	W = 0.000 deg,	P = 30.000 deg,	R = -177.679 deg
};
P[254]{
   GP1:
	UF : 0, UT : 1,		CONFIG : 'N U T, 0, 0, 0',
	X = 1232.321  mm,	Y = 30.350  mm,	Z = -235.021  mm,
	W = 0.000 deg,	P = 30.000 deg,	R = -177.679 deg
};
P[255]{
   GP1:
	UF : 0, UT : 1,		CONFIG : 'N U T, 0, 0, 0',
	X = 1232.240  mm,	Y = 32.348  mm,	Z = -234.989  mm,
	W = 0.000 deg,	P = 30.000 deg,	R = -177.679 deg
};
P[256]{
   GP1:
	UF : 0, UT : 1,		CONFIG : 'N U T, 0, 0, 0',
	X = 1232.159  mm,	Y = 34.346  mm,	Z = -234.956  mm,
	W = 0.000 deg,	P = 30.000 deg,	R = -177.679 deg
};
P[257]{
   GP1:
	UF : 0, UT : 1,		CONFIG : 'N U T, 0, 0, 0',
	X = 1232.078  mm,	Y = 36.344  mm,	Z = -234.924  mm,
	W = 0.000 deg,	P = 30.000 deg,	R = -177.679 deg
};
P[258]{
   GP1:
	UF : 0, UT : 1,		CONFIG : 'N U T, 0, 0, 0',
	X = 1231.997  mm,	Y = 38.342  mm,	Z = -234.892  mm,
	W = 0.000 deg,	P = 30.000 deg,	R = -177.679 deg
};
P[259]{
   GP1:
	UF : 0, UT : 1,		CONFIG : 'N U T, 0, 0, 0',
	X = 1231.916  mm,	Y = 40.341  mm,	Z = -234.859  mm,
	W = 0.000 deg,	P = 30.000 deg,	R = -177.679 deg
};
P[260]{
   GP1:
	UF : 0, UT : 1,		CONFIG : 'N U T, 0, 0, 0',
	X = 1231.835  mm,	Y = 42.339  mm,	Z = -234.827  mm,
	W = 0.000 deg,	P = 30.000 deg,	R = -177.679 deg
};
P[261]{
   GP1:
	UF : 0, UT : 1,		CONFIG : 'N U T, 0, 0, 0',
	X = 1231.754  mm,	Y = 44.337  mm,	Z = -234.795  mm,
	W = 0.000 deg,	P = 30.000 deg,	R = -177.679 deg
};
P[262]{
   GP1:
	UF : 0, UT : 1,		CONFIG : 'N U T, 0, 0, 0',
	X = 1231.673  mm,	Y = 46.335  mm,	Z = -234.762  mm,
	W = 0.000 deg,	P = 30.000 deg,	R = -177.679 deg
};
P[263]{
   GP1:
	UF : 0, UT : 1,		CONFIG : 'N U T, 0, 0, 0',
	X = 1231.592  mm,	Y = 48.333  mm,	Z = -234.730  mm,
	W = 0.000 deg,	P = 30.000 deg,	R = -177.679 deg
};
P[264]{
   GP1:
	UF : 0, UT : 1,		CONFIG : 'N U T, 0, 0, 0',
	X = 1231.511  mm,	Y = 50.331  mm,	Z = -234.698  mm,
	W = 0.000 deg,	P = 30.000 deg,	R = -177.679 deg
};
P[265]{
   GP1:
	UF : 0, UT : 1,		CONFIG : 'N U T, 0, 0, 0',
	X = 1231.430  mm,	Y = 52.329  mm,	Z = -234.665  mm,
	W = 0.000 deg,	P = 30.000 deg,	R = -177.679 deg
};
P[266]{
   GP1:
	UF : 0, UT : 1,		CONFIG : 'N U T, 0, 0, 0',
	X = 1231.349  mm,	Y = 54.327  mm,	Z = -234.633  mm,
	W = 0.000 deg,	P = 30.000 deg,	R = -177.679 deg
};
P[267]{
   GP1:
	UF : 0, UT : 1,		CONFIG : 'N U T, 0, 0, 0',
	X = 1231.268  mm,	Y = 56.325  mm,	Z = -234.601  mm,
	W = 0.000 deg,	P = 30.000 deg,	R = -177.679 deg
};
P[268]{
   GP1:
	UF : 0, UT : 1,		CONFIG : 'N U T, 0, 0, 0',
	X = 1231.187  mm,	Y = 58.323  mm,	Z = -234.568  mm,
	W = 0.000 deg,	P = 30.000 deg,	R = -177.679 deg
};
P[269]{
   GP1:
	UF : 0, UT : 1,		CONFIG : 'N U T, 0, 0, 0',
	X = 1231.106  mm,	Y = 60.322  mm,	Z = -234.536  mm,
	W = 0.000 deg,	P = 30.000 deg,	R = -177.679 deg
};
P[270]{
   GP1:
	UF : 0, UT : 1,		CONFIG : 'N U T, 0, 0, 0',
	X = 1231.025  mm,	Y = 62.320  mm,	Z = -234.504  mm,
	W = 0.000 deg,	P = 30.000 deg,	R = -177.679 deg
};
P[271]{
   GP1:
	UF : 0, UT : 1,		CONFIG : 'N U T, 0, 0, 0',
	X = 1230.944  mm,	Y = 64.318  mm,	Z = -234.472  mm,
	W = 0.000 deg,	P = 30.000 deg,	R = -177.679 deg
};
P[272]{
   GP1:
	UF : 0, UT : 1,		CONFIG : 'N U T, 0, 0, 0',
	X = 1230.863  mm,	Y = 66.316  mm,	Z = -234.439  mm,
	W = 0.000 deg,	P = 30.000 deg,	R = -177.679 deg
};
P[273]{
   GP1:
	UF : 0, UT : 1,		CONFIG : 'N U T, 0, 0, 0',
	X = 1230.782  mm,	Y = 68.314  mm,	Z = -234.407  mm,
	W = 0.000 deg,	P = 30.000 deg,	R = -177.679 deg
};
P[274]{
   GP1:
	UF : 0, UT : 1,		CONFIG : 'N U T, 0, 0, 0',
	X = 1230.701  mm,	Y = 70.312  mm,	Z = -234.375  mm,
	W = 0.000 deg,	P = 30.000 deg,	R = -177.679 deg
};
P[275]{
   GP1:
	UF : 0, UT : 1,		CONFIG : 'N U T, 0, 0, 0',
	X = 1230.620  mm,	Y = 72.310  mm,	Z = -234.342  mm,
	W = 0.000 deg,	P = 30.000 deg,	R = -177.679 deg
};
P[276]{
   GP1:
	UF : 0, UT : 1,		CONFIG : 'N U T, 0, 0, 0',
	X = 1230.539  mm,	Y = 74.308  mm,	Z = -234.310  mm,
	W = 0.000 deg,	P = 30.000 deg,	R = -177.148 deg
};
P[277]{
   GP1:
	UF : 0, UT : 1,		CONFIG : 'N U T, 0, 0, 0',
	X = 1230.458  mm,	Y = 76.306  mm,	Z = -234.278  mm,
	W = 0.000 deg,	P = 30.000 deg,	R = -173.612 deg
};
P[278]{
   GP1:
	UF : 0, UT : 1,		CONFIG : 'N U T, 0, 0, 0',
	X = 1230.377  mm,	Y = 78.304  mm,	Z = -234.245  mm,
	W = 0.000 deg,	P = 30.000 deg,	R = -170.076 deg
};
P[279]{
   GP1:
	UF : 0, UT : 1,		CONFIG : 'N U T, 0, 0, 0',
	X = 1230.296  mm,	Y = 80.303  mm,	Z = -234.213  mm,
	W = 0.000 deg,	P = 30.000 deg,	R = -166.541 deg
};
P[280]{
   GP1:
	UF : 0, UT : 1,		CONFIG : 'N U T, 0, 0, 0',
	X = 1230.215  mm,	Y = 82.301  mm,	Z = -234.181  mm,
	W = 0.000 deg,	P = 30.000 deg,	R = -163.005 deg
};
P[281]{
   GP1:
	UF : 0, UT : 1,		CONFIG : 'N U T, 0, 0, 0',
	X = 1230.134  mm,	Y = 84.299  mm,	Z = -234.148  mm,
	W = 0.000 deg,	P = 30.000 deg,	R = -160.000 deg
};
P[282]{
   GP1:
	UF : 0, UT : 1,		CONFIG : 'N U T, 0, 0, 0',
	X = 1230.120  mm,	Y = 84.652  mm,	Z = -234.143  mm,
	W = 0.000 deg,	P = 30.000 deg,	R = -160.000 deg
};
P[283]{
   GP1:
	UF : 0, UT : 1,		CONFIG : 'N U T, 0, 0, 0',
	X = 1228.982  mm,	Y = 85.808  mm,	Z = -233.863  mm,
	W = 0.000 deg,	P = 30.000 deg,	R = -160.000 deg
};
P[284]{
   GP1:
	UF : 0, UT : 1,		CONFIG : 'N U T, 0, 0, 0',
	X = 1227.599  mm,	Y = 87.213  mm,	Z = -233.523  mm,
	W = 0.000 deg,	P = 30.000 deg,	R = -160.000 deg
};
P[285]{
   GP1:
	UF : 0, UT : 1,		CONFIG : 'N U T, 0, 0, 0',
	X = 1226.216  mm,	Y = 88.617  mm,	Z = -233.183  mm,
	W = 0.000 deg,	P = 30.000 deg,	R = -160.000 deg
};
P[286]{
   GP1:
	UF : 0, UT : 1,		CONFIG : 'N U T, 0, 0, 0',
	X = 1224.833  mm,	Y = 90.021  mm,	Z = -232.843  mm,
	W = 0.000 deg,	P = 30.000 deg,	R = -160.000 deg
};
P[287]{
   GP1:
	UF : 0, UT : 1,		CONFIG : 'N U T, 0, 0, 0',
	X = 1223.451  mm,	Y = 91.426  mm,	Z = -232.502  mm,
	W = 0.000 deg,	P = 30.000 deg,	R = -160.000 deg
};
P[288]{
   GP1:
	UF : 0, UT : 1,		CONFIG : 'N U T, 0, 0, 0',
	X = 1222.068  mm,	Y = 92.830  mm,	Z = -232.162  mm,
	W = 0.000 deg,	P = 30.000 deg,	R = -160.000 deg
};
P[289]{
   GP1:
	UF : 0, UT : 1,		CONFIG : 'N U T, 0, 0, 0',
	X = 1220.685  mm,	Y = 94.235  mm,	Z = -231.822  mm,
	W = 0.000 deg,	P = 30.000 deg,	R = -160.000 deg
};
P[290]{
   GP1:
	UF : 0, UT : 1,		CONFIG : 'N U T, 0, 0, 0',
	X = 1219.302  mm,	Y = 95.639  mm,	Z = -231.482  mm,
	W = 0.000 deg,	P = 30.000 deg,	R = -160.000 deg
};
P[291]{
   GP1:
	UF : 0, UT : 1,		CONFIG : 'N U T, 0, 0, 0',
	X = 1217.920  mm,	Y = 97.043  mm,	Z = -231.142  mm,
	W = 0.000 deg,	P = 30.000 deg,	R = -160.000 deg
};
P[292]{
   GP1:
	UF : 0, UT : 1,		CONFIG : 'N U T, 0, 0, 0',
	X = 1216.537  mm,	Y = 98.448  mm,	Z = -230.802  mm,
	W = 0.000 deg,	P = 30.000 deg,	R = -160.000 deg
};
P[293]{
   GP1:
	UF : 0, UT : 1,		CONFIG : 'N U T, 0, 0, 0',
	X = 1215.154  mm,	Y = 99.852  mm,	Z = -230.462  mm,
	W = 0.000 deg,	P = 30.000 deg,	R = -160.000 deg
};
P[294]{
   GP1:
	UF : 0, UT : 1,		CONFIG : 'N U T, 0, 0, 0',
	X = 1213.771  mm,	Y = 101.257  mm,	Z = -230.122  mm,
	W = 0.000 deg,	P = 30.000 deg,	R = -160.000 deg
};
P[295]{
   GP1:
	UF : 0, UT : 1,		CONFIG : 'N U T, 0, 0, 0',
	X = 1212.389  mm,	Y = 102.661  mm,	Z = -229.782  mm,
	W = 0.000 deg,	P = 30.000 deg,	R = -160.000 deg
};
P[296]{
   GP1:
	UF : 0, UT : 1,		CONFIG : 'N U T, 0, 0, 0',
	X = 1211.006  mm,	Y = 104.065  mm,	Z = -229.442  mm,
	W = 0.000 deg,	P = 30.000 deg,	R = -160.000 deg
};
P[297]{
   GP1:
	UF : 0, UT : 1,		CONFIG : 'N U T, 0, 0, 0',
	X = 1209.623  mm,	Y = 105.470  mm,	Z = -229.102  mm,
	W = 0.000 deg,	P = 30.000 deg,	R = -160.000 deg
};
P[298]{
   GP1:
	UF : 0, UT : 1,		CONFIG : 'N U T, 0, 0, 0',
	X = 1208.240  mm,	Y = 106.874  mm,	Z = -228.762  mm,
	W = 0.000 deg,	P = 30.000 deg,	R = -160.000 deg
};
P[299]{
   GP1:
	UF : 0, UT : 1,		CONFIG : 'N U T, 0, 0, 0',
	X = 1206.858  mm,	Y = 108.279  mm,	Z = -228.422  mm,
	W = 0.000 deg,	P = 30.000 deg,	R = -160.000 deg
};
P[300]{
   GP1:
	UF : 0, UT : 1,		CONFIG : 'N U T, 0, 0, 0',
	X = 1205.475  mm,	Y = 109.683  mm,	Z = -228.082  mm,
	W = 0.000 deg,	P = 30.000 deg,	R = -160.000 deg
};
P[301]{
   GP1:
	UF : 0, UT : 1,		CONFIG : 'N U T, 0, 0, 0',
	X = 1204.092  mm,	Y = 111.087  mm,	Z = -227.741  mm,
	W = 0.000 deg,	P = 30.000 deg,	R = -160.000 deg
};
P[302]{
   GP1:
	UF : 0, UT : 1,		CONFIG : 'N U T, 0, 0, 0',
	X = 1202.709  mm,	Y = 112.492  mm,	Z = -227.401  mm,
	W = 0.000 deg,	P = 30.000 deg,	R = -160.000 deg
};
P[303]{
   GP1:
	UF : 0, UT : 1,		CONFIG : 'N U T, 0, 0, 0',
	X = 1201.327  mm,	Y = 113.896  mm,	Z = -227.061  mm,
	W = 0.000 deg,	P = 30.000 deg,	R = -160.000 deg
};
P[304]{
   GP1:
	UF : 0, UT : 1,		CONFIG : 'N U T, 0, 0, 0',
	X = 1199.944  mm,	Y = 115.301  mm,	Z = -226.721  mm,
	W = 0.000 deg,	P = 30.000 deg,	R = -167.385 deg
};
P[305]{
   GP1:
	UF : 0, UT : 1,		CONFIG : 'N U T, 0, 0, 0',
	X = 1198.561  mm,	Y = 116.705  mm,	Z = -226.381  mm,
	W = 0.000 deg,	P = 30.000 deg,	R = -171.436 deg
};
P[306]{
   GP1:
	UF : 0, UT : 1,		CONFIG : 'N U T, 0, 0, 0',
	X = 1197.178  mm,	Y = 118.110  mm,	Z = -226.041  mm,
	W = 0.000 deg,	P = 30.000 deg,	R = -175.487 deg
};
P[307]{
   GP1:
	UF : 0, UT : 1,		CONFIG : 'N U T, 0, 0, 0',
	X = 1195.796  mm,	Y = 119.514  mm,	Z = -225.701  mm,
	W = 0.000 deg,	P = 30.000 deg,	R = -179.537 deg
};
P[308]{
   GP1:
	UF : 0, UT : 1,		CONFIG : 'N U T, 0, 0, 0',
	X = 1194.413  mm,	Y = 120.918  mm,	Z = -225.361  mm,
	W = 0.000 deg,	P = 30.000 deg,	R = 179.746 deg
};
P[309]{
   GP1:
	UF : 0, UT : 1,		CONFIG : 'N U T, 0, 0, 0',
	X = 1194.315  mm,	Y = 121.018  mm,	Z = -225.337  mm,
	W = 0.000 deg,	P = 30.000 deg,	R = 179.746 deg
};
P[310]{
   GP1:
	UF : 0, UT : 1,		CONFIG : 'N U T, 0, 0, 0',
	X = 1194.323  mm,	Y = 122.876  mm,	Z = -225.326  mm,
	W = 0.000 deg,	P = 30.000 deg,	R = 179.746 deg
};
P[311]{
   GP1:
	UF : 0, UT : 1,		CONFIG : 'N U T, 0, 0, 0',
	X = 1194.332  mm,	Y = 124.876  mm,	Z = -225.314  mm,
	W = 0.000 deg,	P = 30.000 deg,	R = 179.746 deg
};
P[312]{
   GP1:
	UF : 0, UT : 1,		CONFIG : 'N U T, 0, 0, 0',
	X = 1194.341  mm,	Y = 126.876  mm,	Z = -225.303  mm,
	W = 0.000 deg,	P = 30.000 deg,	R = 179.746 deg
};
P[313]{
   GP1:
	UF : 0, UT : 1,		CONFIG : 'N U T, 0, 0, 0',
	X = 1194.350  mm,	Y = 128.876  mm,	Z = -225.291  mm,
	W = 0.000 deg,	P = 30.000 deg,	R = 179.746 deg
};
P[314]{
   GP1:
	UF : 0, UT : 1,		CONFIG : 'N U T, 0, 0, 0',
	X = 1194.359  mm,	Y = 130.876  mm,	Z = -225.279  mm,
	W = 0.000 deg,	P = 30.000 deg,	R = 179.746 deg
};
P[315]{
   GP1:
	UF : 0, UT : 1,		CONFIG : 'N U T, 0, 0, 0',
	X = 1194.368  mm,	Y = 132.876  mm,	Z = -225.268  mm,
	W = 0.000 deg,	P = 30.000 deg,	R = 179.746 deg
};
P[316]{
   GP1:
	UF : 0, UT : 1,		CONFIG : 'N U T, 0, 0, 0',
	X = 1194.377  mm,	Y = 134.876  mm,	Z = -225.256  mm,
	W = 0.000 deg,	P = 30.000 deg,	R = 179.746 deg
};
P[317]{
   GP1:
	UF : 0, UT : 1,		CONFIG : 'N U T, 0, 0, 0',
	X = 1194.385  mm,	Y = 136.876  mm,	Z = -225.244  mm,
	W = 0.000 deg,	P = 30.000 deg,	R = 179.746 deg
};
P[318]{
   GP1:
	UF : 0, UT : 1,		CONFIG : 'N U T, 0, 0, 0',
	X = 1194.394  mm,	Y = 138.876  mm,	Z = -225.233  mm,
	W = 0.000 deg,	P = 30.000 deg,	R = 179.746 deg
};
P[319]{
   GP1:
	UF : 0, UT : 1,		CONFIG : 'N U T, 0, 0, 0',
	X = 1194.403  mm,	Y = 140.876  mm,	Z = -225.221  mm,
	W = 0.000 deg,	P = 30.000 deg,	R = 179.746 deg
};
P[320]{
   GP1:
	UF : 0, UT : 1,		CONFIG : 'N U T, 0, 0, 0',
	X = 1194.412  mm,	Y = 142.876  mm,	Z = -225.209  mm,
	W = 0.000 deg,	P = 30.000 deg,	R = 179.746 deg
};
P[321]{
   GP1:
	UF : 0, UT : 1,		CONFIG : 'N U T, 0, 0, 0',
	X = 1194.421  mm,	Y = 144.876  mm,	Z = -225.198  mm,
	W = 0.000 deg,	P = 30.000 deg,	R = 179.746 deg
};
P[322]{
   GP1:
	UF : 0, UT : 1,		CONFIG : 'N U T, 0, 0, 0',
	X = 1194.430  mm,	Y = 146.876  mm,	Z = -225.186  mm,
	W = 0.000 deg,	P = 30.000 deg,	R = 179.746 deg
};
P[323]{
   GP1:
	UF : 0, UT : 1,		CONFIG : 'N U T, 0, 0, 0',
	X = 1194.438  mm,	Y = 148.876  mm,	Z = -225.175  mm,
	W = 0.000 deg,	P = 30.000 deg,	R = 179.746 deg
};
P[324]{
   GP1:
	UF : 0, UT : 1,		CONFIG : 'N U T, 0, 0, 0',
	X = 1194.447  mm,	Y = 150.875  mm,	Z = -225.163  mm,
	W = 0.000 deg,	P = 30.000 deg,	R = 179.746 deg
};
P[325]{
   GP1:
	UF : 0, UT : 1,		CONFIG : 'N U T, 0, 0, 0',
	X = 1194.456  mm,	Y = 152.875  mm,	Z = -225.151  mm,
	W = 0.000 deg,	P = 30.000 deg,	R = 179.746 deg
};
P[326]{
   GP1:
	UF : 0, UT : 1,		CONFIG : 'N U T, 0, 0, 0',
	X = 1194.465  mm,	Y = 154.875  mm,	Z = -225.140  mm,
	W = 0.000 deg,	P = 30.000 deg,	R = 179.746 deg
};
P[327]{
   GP1:
	UF : 0, UT : 1,		CONFIG : 'N U T, 0, 0, 0',
	X = 1194.474  mm,	Y = 156.875  mm,	Z = -225.128  mm,
	W = 0.000 deg,	P = 30.000 deg,	R = 179.746 deg
};
P[328]{
   GP1:
	UF : 0, UT : 1,		CONFIG : 'N U T, 0, 0, 0',
	X = 1194.483  mm,	Y = 158.875  mm,	Z = -225.116  mm,
	W = 0.000 deg,	P = 30.000 deg,	R = 179.746 deg
};
P[329]{
   GP1:
	UF : 0, UT : 1,		CONFIG : 'N U T, 0, 0, 0',
	X = 1194.492  mm,	Y = 160.875  mm,	Z = -225.105  mm,
	W = 0.000 deg,	P = 30.000 deg,	R = 179.746 deg
};
P[330]{
   GP1:
	UF : 0, UT : 1,		CONFIG : 'N U T, 0, 0, 0',
	X = 1194.500  mm,	Y = 162.875  mm,	Z = -225.093  mm,
	W = 0.000 deg,	P = 30.000 deg,	R = 179.746 deg
};
P[331]{
   GP1:
	UF : 0, UT : 1,		CONFIG : 'N U T, 0, 0, 0',
	X = 1194.509  mm,	Y = 164.875  mm,	Z = -225.081  mm,
	W = 0.000 deg,	P = 30.000 deg,	R = 179.746 deg
};
P[332]{
   GP1:
	UF : 0, UT : 1,		CONFIG : 'N U T, 0, 0, 0',
	X = 1194.518  mm,	Y = 166.875  mm,	Z = -225.070  mm,
	W = 0.000 deg,	P = 30.000 deg,	R = 179.746 deg
};
P[333]{
   GP1:
	UF : 0, UT : 1,		CONFIG : 'N U T, 0, 0, 0',
	X = 1194.527  mm,	Y = 168.875  mm,	Z = -225.058  mm,
	W = 0.000 deg,	P = 30.000 deg,	R = 179.746 deg
};
P[334]{
   GP1:
	UF : 0, UT : 1,		CONFIG : 'N U T, 0, 0, 0',
	X = 1194.536  mm,	Y = 170.875  mm,	Z = -225.046  mm,
	W = 0.000 deg,	P = 30.000 deg,	R = 179.746 deg
};
P[335]{
   GP1:
	UF : 0, UT : 1,		CONFIG : 'N U T, 0, 0, 0',
	X = 1194.545  mm,	Y = 172.875  mm,	Z = -225.035  mm,
	W = 0.000 deg,	P = 30.000 deg,	R = 172.127 deg
};
P[336]{
   GP1:
	UF : 0, UT : 1,		CONFIG : 'N U T, 0, 0, 0',
	X = 1194.554  mm,	Y = 174.875  mm,	Z = -225.023  mm,
	W = 0.000 deg,	P = 30.000 deg,	R = 168.178 deg
};
P[337]{
   GP1:
	UF : 0, UT : 1,		CONFIG : 'N U T, 0, 0, 0',
	X = 1194.562  mm,	Y = 176.875  mm,	Z = -225.011  mm,
	W = 0.000 deg,	P = 30.000 deg,	R = 164.228 deg
};
P[338]{
   GP1:
	UF : 0, UT : 1,		CONFIG : 'N U T, 0, 0, 0',
	X = 1194.571  mm,	Y = 178.875  mm,	Z = -225.000  mm,
	W = 0.000 deg,	P = 30.000 deg,	R = 160.279 deg
};
P[339]{
   GP1:
	UF : 0, UT : 1,		CONFIG : 'N U T, 0, 0, 0',
	X = 1194.577  mm,	Y = 180.219  mm,	Z = -224.992  mm,
	W = 0.000 deg,	P = 30.000 deg,	R = 160.000 deg
};
P[340]{
   GP1:
	UF : 0, UT : 1,		CONFIG : 'N U T, 0, 0, 0',
	X = 1195.024  mm,	Y = 180.686  mm,	Z = -225.099  mm,
	W = 0.000 deg,	P = 30.000 deg,	R = 160.000 deg
};
P[341]{
   GP1:
	UF : 0, UT : 1,		CONFIG : 'N U T, 0, 0, 0',
	X = 1196.389  mm,	Y = 182.112  mm,	Z = -225.426  mm,
	W = 0.000 deg,	P = 30.000 deg,	R = 160.000 deg
};
P[342]{
   GP1:
	UF : 0, UT : 1,		CONFIG : 'N U T, 0, 0, 0',
	X = 1197.753  mm,	Y = 183.537  mm,	Z = -225.753  mm,
	W = 0.000 deg,	P = 30.000 deg,	R = 160.000 deg
};
P[343]{
   GP1:
	UF : 0, UT : 1,		CONFIG : 'N U T, 0, 0, 0',
	X = 1199.117  mm,	Y = 184.962  mm,	Z = -226.080  mm,
	W = 0.000 deg,	P = 30.000 deg,	R = 160.000 deg
};
P[344]{
   GP1:
	UF : 0, UT : 1,		CONFIG : 'N U T, 0, 0, 0',
	X = 1200.482  mm,	Y = 186.387  mm,	Z = -226.407  mm,
	W = 0.000 deg,	P = 30.000 deg,	R = 160.000 deg
};
P[345]{
   GP1:
	UF : 0, UT : 1,		CONFIG : 'N U T, 0, 0, 0',
	X = 1201.846  mm,	Y = 187.813  mm,	Z = -226.734  mm,
	W = 0.000 deg,	P = 30.000 deg,	R = 160.000 deg
};
P[346]{
   GP1:
	UF : 0, UT : 1,		CONFIG : 'N U T, 0, 0, 0',
	X = 1203.211  mm,	Y = 189.238  mm,	Z = -227.061  mm,
	W = 0.000 deg,	P = 30.000 deg,	R = 160.000 deg
};
P[347]{
   GP1:
	UF : 0, UT : 1,		CONFIG : 'N U T, 0, 0, 0',
	X = 1204.575  mm,	Y = 190.663  mm,	Z = -227.388  mm,
	W = 0.000 deg,	P = 30.000 deg,	R = 160.000 deg
};
P[348]{
   GP1:
	UF : 0, UT : 1,		CONFIG : 'N U T, 0, 0, 0',
	X = 1205.939  mm,	Y = 192.089  mm,	Z = -227.716  mm,
	W = 0.000 deg,	P = 30.000 deg,	R = 160.000 deg
};
P[349]{
   GP1:
	UF : 0, UT : 1,		CONFIG : 'N U T, 0, 0, 0',
	X = 1207.304  mm,	Y = 193.514  mm,	Z = -228.043  mm,
	W = 0.000 deg,	P = 30.000 deg,	R = 160.000 deg
};
P[350]{
   GP1:
	UF : 0, UT : 1,		CONFIG : 'N U T, 0, 0, 0',
	X = 1208.668  mm,	Y = 194.939  mm,	Z = -228.370  mm,
	W = 0.000 deg,	P = 30.000 deg,	R = 160.000 deg
};
P[351]{
   GP1:
	UF : 0, UT : 1,		CONFIG : 'N U T, 0, 0, 0',
	X = 1210.033  mm,	Y = 196.364  mm,	Z = -228.697  mm,
	W = 0.000 deg,	P = 30.000 deg,	R = 160.000 deg
};
P[352]{
   GP1:
	UF : 0, UT : 1,		CONFIG : 'N U T, 0, 0, 0',
	X = 1211.397  mm,	Y = 197.790  mm,	Z = -229.024  mm,
	W = 0.000 deg,	P = 30.000 deg,	R = 160.000 deg
};
P[353]{
   GP1:
	UF : 0, UT : 1,		CONFIG : 'N U T, 0, 0, 0',
	X = 1212.761  mm,	Y = 199.215  mm,	Z = -229.351  mm,
	W = 0.000 deg,	P = 30.000 deg,	R = 160.000 deg
};
P[354]{
   GP1:
	UF : 0, UT : 1,		CONFIG : 'N U T, 0, 0, 0',
	X = 1214.126  mm,	Y = 200.640  mm,	Z = -229.678  mm,
	W = 0.000 deg,	P = 30.000 deg,	R = 160.000 deg
};
P[355]{
   GP1:
	UF : 0, UT : 1,		CONFIG : 'N U T, 0, 0, 0',
	X = 1215.490  mm,	Y = 202.065  mm,	Z = -230.005  mm,
	W = 0.000 deg,	P = 30.000 deg,	R = 160.000 deg
};
P[356]{
   GP1:
	UF : 0, UT : 1,		CONFIG : 'N U T, 0, 0, 0',
	X = 1216.855  mm,	Y = 203.491  mm,	Z = -230.332  mm,
	W = 0.000 deg,	P = 30.000 deg,	R = 160.000 deg
};
P[357]{
   GP1:
	UF : 0, UT : 1,		CONFIG : 'N U T, 0, 0, 0',
	X = 1218.219  mm,	Y = 204.916  mm,	Z = -230.659  mm,
	W = 0.000 deg,	P = 30.000 deg,	R = 160.000 deg
};
P[358]{
   GP1:
	UF : 0, UT : 1,		CONFIG : 'N U T, 0, 0, 0',
	X = 1219.584  mm,	Y = 206.341  mm,	Z = -230.986  mm,
	W = 0.000 deg,	P = 30.000 deg,	R = 160.000 deg
};
P[359]{
   GP1:
	UF : 0, UT : 1,		CONFIG : 'N U T, 0, 0, 0',
	X = 1220.948  mm,	Y = 207.767  mm,	Z = -231.313  mm,
	W = 0.000 deg,	P = 30.000 deg,	R = 160.000 deg
};
P[360]{
   GP1:
	UF : 0, UT : 1,		CONFIG : 'N U T, 0, 0, 0',
	X = 1222.312  mm,	Y = 209.192  mm,	Z = -231.641  mm,
	W = 0.000 deg,	P = 30.000 deg,	R = 160.000 deg
};
P[361]{
   GP1:
	UF : 0, UT : 1,		CONFIG : 'N U T, 0, 0, 0',
	X = 1223.677  mm,	Y = 210.617  mm,	Z = -231.968  mm,
	W = 0.000 deg,	P = 30.000 deg,	R = 165.434 deg
};
P[362]{
   GP1:
	UF : 0, UT : 1,		CONFIG : 'N U T, 0, 0, 0',
	X = 1225.041  mm,	Y = 212.042  mm,	Z = -232.295  mm,
	W = 0.000 deg,	P = 30.000 deg,	R = 169.527 deg
};
P[363]{
   GP1:
	UF : 0, UT : 1,		CONFIG : 'N U T, 0, 0, 0',
	X = 1226.406  mm,	Y = 213.468  mm,	Z = -232.622  mm,
	W = 0.000 deg,	P = 30.000 deg,	R = 173.619 deg
};
P[364]{
   GP1:
	UF : 0, UT : 1,		CONFIG : 'N U T, 0, 0, 0',
	X = 1227.770  mm,	Y = 214.893  mm,	Z = -232.949  mm,
	W = 0.000 deg,	P = 30.000 deg,	R = 177.712 deg
};
P[365]{
   GP1:
	UF : 0, UT : 1,		CONFIG : 'N U T, 0, 0, 0',
	X = 1229.134  mm,	Y = 216.318  mm,	Z = -233.276  mm,
	W = 0.000 deg,	P = 30.000 deg,	R = -179.536 deg
};
P[366]{
   GP1:
	UF : 0, UT : 1,		CONFIG : 'N U T, 0, 0, 0',
	X = 1229.368  mm,	Y = 216.562  mm,	Z = -233.332  mm,
	W = 0.000 deg,	P = 30.000 deg,	R = -179.536 deg
};
P[367]{
   GP1:
	UF : 0, UT : 1,		CONFIG : 'N U T, 0, 0, 0',
	X = 1229.354  mm,	Y = 218.220  mm,	Z = -233.324  mm,
	W = 0.000 deg,	P = 30.000 deg,	R = -179.536 deg
};
P[368]{
   GP1:
	UF : 0, UT : 1,		CONFIG : 'N U T, 0, 0, 0',
	X = 1229.338  mm,	Y = 220.220  mm,	Z = -233.314  mm,
	W = 0.000 deg,	P = 30.000 deg,	R = -179.536 deg
};
P[369]{
   GP1:
	UF : 0, UT : 1,		CONFIG : 'N U T, 0, 0, 0',
	X = 1229.322  mm,	Y = 222.220  mm,	Z = -233.304  mm,
	W = 0.000 deg,	P = 30.000 deg,	R = -179.536 deg
};
P[370]{
   GP1:
	UF : 0, UT : 1,		CONFIG : 'N U T, 0, 0, 0',
	X = 1229.306  mm,	Y = 224.220  mm,	Z = -233.295  mm,
	W = 0.000 deg,	P = 30.000 deg,	R = -179.536 deg
};
P[371]{
   GP1:
	UF : 0, UT : 1,		CONFIG : 'N U T, 0, 0, 0',
	X = 1229.289  mm,	Y = 226.219  mm,	Z = -233.285  mm,
	W = 0.000 deg,	P = 30.000 deg,	R = -179.536 deg
};
P[372]{
   GP1:
	UF : 0, UT : 1,		CONFIG : 'N U T, 0, 0, 0',
	X = 1229.273  mm,	Y = 228.219  mm,	Z = -233.275  mm,
	W = 0.000 deg,	P = 30.000 deg,	R = -179.536 deg
};
P[373]{
   GP1:
	UF : 0, UT : 1,		CONFIG : 'N U T, 0, 0, 0',
	X = 1229.271  mm,	Y = 228.561  mm,	Z = -233.274  mm,
	W = 0.000 deg,	P = 30.000 deg,	R = -179.536 deg
};
/END
